LIN {X 0,Y 204.724,Z 772.28,A -85,B 0,C 180,E1 -21058.033,E2 -21058.033} C_VEL
LIN {X 0,Y 204.875,Z 767.063,A -85,B 0,C 180,E1 -21060.983,E2 -21060.983} C_VEL
LIN {X 0,Y 205.148,Z 761.459,A -85,B 0,C 180,E1 -21063.437,E2 -21063.437} C_VEL
LIN {X 0,Y 205.482,Z 754.231,A -85,B 0,C 180,E1 -21065.889,E2 -21065.889} C_VEL
LIN {X 0,Y 205.8,Z 746.691,A -85,B 0,C 180,E1 -21067.962,E2 -21067.962} C_VEL
LIN {X 0,Y 206.336,Z 737.426,A -85,B 0,C 180,E1 -21070.053,E2 -21070.053} C_VEL
LIN {X 0,Y 206.914,Z 727.818,A -85,B 0,C 180,E1 -21071.759,E2 -21071.759} C_VEL
LIN {X 0,Y 207.533,Z 717.475,A -85,B 0,C 180,E1 -21073.214,E2 -21073.214} C_VEL
LIN {X 0,Y 208.014,Z 706.264,A -85,B 0,C 180,E1 -21074.429,E2 -21074.429} C_VEL
LIN {X 0,Y 208.451,Z 692.158,A -85,B 0,C 180,E1 -21075.46,E2 -21075.46} C_VEL
LIN {X 0,Y 209.728,Z 644.97,A -85,B 0,C 180,E1 -21078.295,E2 -21078.295} C_VEL
LIN {X 0,Y 208.127,Z 622.961,A -85,B 0,C 180,E1 -21079.605,E2 -21079.605} C_VEL
LIN {X 0,Y 208.064,Z 617.38,A -85,B 0,C 180,E1 -21079.999,E2 -21079.999} C_VEL
LIN {X 0,Y 210.025,Z 597.2,A -85,B 0,C 180,E1 -21085.376,E2 -21085.376} C_VEL
LIN {X 0,Y 211.523,Z 584.285,A -85,B 0,C 180,E1 -21088.801,E2 -21088.801} C_VEL
LIN {X 0,Y 211.615,Z 582.311,A -85,B 0,C 180,E1 -21089.332,E2 -21089.332} C_VEL
LIN {X 0,Y 207.961,Z 564.134,A -85,B 0,C 180,E1 -21094.49,E2 -21094.49} C_VEL
LIN {X 0,Y 206.873,Z 558.873,A -85,B 0,C 180,E1 -21096.097,E2 -21096.097} C_VEL
LIN {X 0,Y 206.676,Z 558.686,A -85,B 0,C 180,E1 -21100.248,E2 -21100.248} C_VEL
LIN {X 0,Y 206.636,Z 558.719,A -85,B 0,C 180,E1 -21105.581,E2 -21105.581} C_VEL
LIN {X 0,Y 206.669,Z 558.926,A -85,B 0,C 180,E1 -21108.36,E2 -21108.36} C_VEL
LIN {X 0,Y 206.993,Z 560.154,A -85,B 0,C 180,E1 -21108.764,E2 -21108.764} C_VEL
LIN {X 0,Y 208.656,Z 562.795,A -85,B 0,C 180,E1 -21109.302,E2 -21109.302} C_VEL
LIN {X 0,Y 209.688,Z 564.185,A -85,B 0,C 180,E1 -21109.608,E2 -21109.608} C_VEL
LIN {X 0,Y 217.052,Z 575.841,A -85,B 0,C 180,E1 -21111.739,E2 -21111.739} C_VEL
LIN {X 0,Y 223.541,Z 588.628,A -85,B 0,C 180,E1 -21113.553,E2 -21113.553} C_VEL
LIN {X 0,Y 229.847,Z 603.206,A -85,B 0,C 180,E1 -21115.261,E2 -21115.261} C_VEL
LIN {X 0,Y 230.908,Z 606.056,A -85,B 0,C 180,E1 -21115.551,E2 -21115.551} C_VEL
LIN {X 0,Y 228.358,Z 664.194,A -85,B 0,C 180,E1 -21117.332,E2 -21117.332} C_VEL
LIN {X 0,Y 227.04,Z 677.769,A -85,B 0,C 180,E1 -21118.087,E2 -21118.087} C_VEL
LIN {X 0,Y 225.244,Z 690.404,A -85,B 0,C 180,E1 -21119.143,E2 -21119.143} C_VEL
LIN {X 0,Y 223.064,Z 702.192,A -85,B 0,C 180,E1 -21120.507,E2 -21120.507} C_VEL
LIN {X 0,Y 220.496,Z 713.529,A -85,B 0,C 180,E1 -21122.214,E2 -21122.214} C_VEL
LIN {X 0,Y 217.847,Z 723.743,A -85,B 0,C 180,E1 -21124.18,E2 -21124.18} C_VEL
LIN {X 0,Y 215.4,Z 732.864,A -85,B 0,C 180,E1 -21126.428,E2 -21126.428} C_VEL
LIN {X 0,Y 212.502,Z 741.807,A -85,B 0,C 180,E1 -21129.173,E2 -21129.173} C_VEL
LIN {X 0,Y 210.099,Z 748.972,A -85,B 0,C 180,E1 -21131.974,E2 -21131.974} C_VEL
LIN {X 0,Y 208.48,Z 753.802,A -85,B 0,C 180,E1 -21134.353,E2 -21134.353} C_VEL
LIN {X 0,Y 206.851,Z 758.495,A -85,B 0,C 180,E1 -21137.24,E2 -21137.24} C_VEL
LIN {X 0,Y 205.728,Z 762.077,A -85,B 0,C 180,E1 -21140.164,E2 -21140.164} C_VEL
LIN {X 0,Y 205.202,Z 763.927,A -85,B 0,C 180,E1 -21142.124,E2 -21142.124} C_VEL
LIN {X 0,Y 204.775,Z 765.519,A -85,B 0,C 180,E1 -21144.445,E2 -21144.445} C_VEL
LIN {X 0,Y 204.5,Z 766.916,A -85,B 0,C 180,E1 -21148.029,E2 -21148.029} C_VEL
LIN {X 0,Y 204.499,Z 767.144,A -85,B 0,C 180,E1 -21149.998,E2 -21149.998} C_VEL
LIN {X 0,Y 204.499,Z 766.951,A -85,B 0,C 180,E1 -21151.968,E2 -21151.968} C_VEL
LIN {X 0,Y 204.773,Z 765.603,A -85,B 0,C 180,E1 -21155.551,E2 -21155.551} C_VEL
LIN {X 0,Y 205.2,Z 764.046,A -85,B 0,C 180,E1 -21157.872,E2 -21157.872} C_VEL
LIN {X 0,Y 206.039,Z 761.177,A -85,B 0,C 180,E1 -21160.811,E2 -21160.811} C_VEL
LIN {X 0,Y 207.303,Z 757.284,A -85,B 0,C 180,E1 -21163.726,E2 -21163.726} C_VEL
LIN {X 0,Y 209.022,Z 752.264,A -85,B 0,C 180,E1 -21166.605,E2 -21166.605} C_VEL
LIN {X 0,Y 211.15,Z 745.94,A -85,B 0,C 180,E1 -21169.44,E2 -21169.44} C_VEL
LIN {X 0,Y 213.861,Z 738.019,A -85,B 0,C 180,E1 -21172.203,E2 -21172.203} C_VEL
LIN {X 0,Y 216.152,Z 730.125,A -85,B 0,C 180,E1 -21174.439,E2 -21174.439} C_VEL
LIN {X 0,Y 218.883,Z 720.101,A -85,B 0,C 180,E1 -21176.711,E2 -21176.711} C_VEL
LIN {X 0,Y 221.635,Z 709.007,A -85,B 0,C 180,E1 -21178.658,E2 -21178.658} C_VEL
LIN {X 0,Y 224.044,Z 698.121,A -85,B 0,C 180,E1 -21180.124,E2 -21180.124} C_VEL
LIN {X 0,Y 226.034,Z 686.085,A -85,B 0,C 180,E1 -21181.384,E2 -21181.384} C_VEL
LIN {X 0,Y 227.663,Z 673.169,A -85,B 0,C 180,E1 -21182.342,E2 -21182.342} C_VEL
LIN {X 0,Y 228.776,Z 659.415,A -85,B 0,C 180,E1 -21182.971,E2 -21182.971} C_VEL
LIN {X 0,Y 231.03,Z 606.183,A -85,B 0,C 180,E1 -21184.57,E2 -21184.57} C_VEL
LIN {X 0,Y 225.138,Z 592.104,A -85,B 0,C 180,E1 -21186.161,E2 -21186.161} C_VEL
LIN {X 0,Y 217.878,Z 577.227,A -85,B 0,C 180,E1 -21188.189,E2 -21188.189} C_VEL
LIN {X 0,Y 211.372,Z 566.808,A -85,B 0,C 180,E1 -21190.051,E2 -21190.051} C_VEL
LIN {X 0,Y 208.94,Z 563.085,A -85,B 0,C 180,E1 -21190.784,E2 -21190.784} C_VEL
LIN {X 0,Y 207.22,Z 560.726,A -85,B 0,C 180,E1 -21191.305,E2 -21191.305} C_VEL
LIN {X 0,Y 206.643,Z 558.739,A -85,B 0,C 180,E1 -21191.562,E2 -21191.562} C_VEL
LIN {X 0,Y 206.656,Z 558.72,A -85,B 0,C 180,E1 -21195.573,E2 -21195.573} C_VEL
LIN {X 0,Y 206.699,Z 558.712,A -85,B 0,C 180,E1 -21199.757,E2 -21199.757} C_VEL
LIN {X 0,Y 206.719,Z 558.701,A -85,B 0,C 180,E1 -21202.268,E2 -21202.268} C_VEL
LIN {X 0,Y 206.705,Z 558.728,A -85,B 0,C 180,E1 -21207.043,E2 -21207.043} C_VEL
LIN {X 0,Y 206.761,Z 558.716,A -85,B 0,C 180,E1 -21212.095,E2 -21212.095} C_VEL
LIN {X 0,Y 206.78,Z 558.717,A -85,B 0,C 180,E1 -21216.583,E2 -21216.583} C_VEL
LIN {X 0,Y 206.87,Z 558.707,A -85,B 0,C 180,E1 -21222.196,E2 -21222.196} C_VEL
LIN {X 0,Y 206.907,Z 558.71,A -85,B 0,C 180,E1 -21226.245,E2 -21226.245} C_VEL
LIN {X 0,Y 207.099,Z 558.667,A -85,B 0,C 180,E1 -21230.231,E2 -21230.231} C_VEL
LIN {X 0,Y 207.172,Z 558.672,A -85,B 0,C 180,E1 -21232.201,E2 -21232.201} C_VEL
LIN {X 0,Y 207.377,Z 558.637,A -85,B 0,C 180,E1 -21238.058,E2 -21238.058} C_VEL
LIN {X 0,Y 207.513,Z 558.637,A -85,B 0,C 180,E1 -21240,E2 -21240} C_VEL
LIN {X 0,Y 207.081,Z 558.67,A -85,B 0,C 180,E1 -21243.892,E2 -21243.892} C_VEL
LIN {X 0,Y 207.182,Z 558.674,A -85,B 0,C 180,E1 -21247.798,E2 -21247.798} C_VEL
LIN {X 0,Y 206.977,Z 558.693,A -85,B 0,C 180,E1 -21251.755,E2 -21251.755} C_VEL
LIN {X 0,Y 206.86,Z 558.701,A -85,B 0,C 180,E1 -21255.771,E2 -21255.771} C_VEL
LIN {X 0,Y 206.794,Z 558.723,A -85,B 0,C 180,E1 -21259.868,E2 -21259.868} C_VEL
LIN {X 0,Y 206.758,Z 558.732,A -85,B 0,C 180,E1 -21264.073,E2 -21264.073} C_VEL
LIN {X 0,Y 206.731,Z 558.734,A -85,B 0,C 180,E1 -21268.421,E2 -21268.421} C_VEL
LIN {X 0,Y 206.695,Z 558.729,A -85,B 0,C 180,E1 -21271.075,E2 -21271.075} C_VEL
LIN {X 0,Y 206.05,Z 558.819,A -85,B 0,C 180,E1 -21272.703,E2 -21272.703} C_VEL
LIN {X 0,Y 203.254,Z 559.173,A -85,B 0,C 180,E1 -21275.362,E2 -21275.362} C_VEL
LIN {X 0,Y 199.998,Z 559.573,A -85,B 0,C 180,E1 -21278.655,E2 -21278.655} C_VEL
LIN {X 0,Y 199.629,Z 559.607,A -85,B 0,C 180,E1 -21279.797,E2 -21279.797} C_VEL
LIN {X 0,Y 199.665,Z 559.81,A -85,B 0,C 180,E1 -21283.274,E2 -21283.274} C_VEL
LIN {X 0,Y 201.361,Z 565.661,A -85,B 0,C 180,E1 -21286.98,E2 -21286.98} C_VEL
LIN {X 0,Y 203.872,Z 570.229,A -85,B 0,C 180,E1 -21287.939,E2 -21287.939} C_VEL
LIN {X 0,Y 209.554,Z 580.484,A -85,B 0,C 180,E1 -21289.769,E2 -21289.769} C_VEL
LIN {X 0,Y 215.497,Z 592.713,A -85,B 0,C 180,E1 -21291.594,E2 -21291.594} C_VEL
LIN {X 0,Y 221.774,Z 607.31,A -85,B 0,C 180,E1 -21293.438,E2 -21293.438} C_VEL
LIN {X 0,Y 222.893,Z 610.664,A -85,B 0,C 180,E1 -21293.781,E2 -21293.781} C_VEL
LIN {X 0,Y 224.53,Z 623.993,A -85,B 0,C 180,E1 -21294.597,E2 -21294.597} C_VEL
LIN {X 0,Y 222.139,Z 674.383,A -85,B 0,C 180,E1 -21296.153,E2 -21296.153} C_VEL
LIN {X 0,Y 220.753,Z 687.704,A -85,B 0,C 180,E1 -21296.876,E2 -21296.876} C_VEL
LIN {X 0,Y 218.746,Z 699.995,A -85,B 0,C 180,E1 -21297.853,E2 -21297.853} C_VEL
LIN {X 0,Y 216.331,Z 712.2,A -85,B 0,C 180,E1 -21299.227,E2 -21299.227} C_VEL
LIN {X 0,Y 213.511,Z 723.759,A -85,B 0,C 180,E1 -21300.956,E2 -21300.956} C_VEL
LIN {X 0,Y 210.62,Z 734.171,A -85,B 0,C 180,E1 -21302.96,E2 -21302.96} C_VEL
LIN {X 0,Y 208.015,Z 742.689,A -85,B 0,C 180,E1 -21305.021,E2 -21305.021} C_VEL
LIN {X 0,Y 205.094,Z 751.926,A -85,B 0,C 180,E1 -21307.858,E2 -21307.858} C_VEL
LIN {X 0,Y 202.534,Z 759.353,A -85,B 0,C 180,E1 -21310.754,E2 -21310.754} C_VEL
LIN {X 0,Y 200.516,Z 765.318,A -85,B 0,C 180,E1 -21313.718,E2 -21313.718} C_VEL
LIN {X 0,Y 199.003,Z 770.036,A -85,B 0,C 180,E1 -21316.731,E2 -21316.731} C_VEL
LIN {X 0,Y 198.024,Z 773.649,A -85,B 0,C 180,E1 -21319.78,E2 -21319.78} C_VEL
LIN {X 0,Y 197.589,Z 775.512,A -85,B 0,C 180,E1 -21321.822,E2 -21321.822} C_VEL
LIN {X 0,Y 197.34,Z 776.909,A -85,B 0,C 180,E1 -21323.869,E2 -21323.869} C_VEL
LIN {X 0,Y 197.235,Z 778.517,A -85,B 0,C 180,E1 -21327.96,E2 -21327.96} C_VEL
LIN {X 0,Y 197.324,Z 778.731,A -85,B 0,C 180,E1 -21330.002,E2 -21330.002} C_VEL
LIN {X 0,Y 197.586,Z 777.91,A -85,B 0,C 180,E1 -21334.081,E2 -21334.081} C_VEL
LIN {X 0,Y 197.728,Z 777.713,A -85,B 0,C 180,E1 -21335.054,E2 -21335.054} C_VEL
LIN {X 0,Y 198.017,Z 780.538,A -85,B 0,C 180,E1 -21338.163,E2 -21338.163} C_VEL
LIN {X 0,Y 198.49,Z 781.851,A -85,B 0,C 180,E1 -21340.199,E2 -21340.199} C_VEL
LIN {X 0,Y 199.342,Z 782.728,A -85,B 0,C 180,E1 -21342.214,E2 -21342.214} C_VEL
LIN {X 0,Y 200.485,Z 783.034,A -85,B 0,C 180,E1 -21344.206,E2 -21344.206} C_VEL
LIN {X 0,Y 201.844,Z 782.917,A -85,B 0,C 180,E1 -21346.175,E2 -21346.175} C_VEL
LIN {X 0,Y 203.512,Z 782.403,A -85,B 0,C 180,E1 -21348.109,E2 -21348.109} C_VEL
LIN {X 0,Y 205.451,Z 781.417,A -85,B 0,C 180,E1 -21350.005,E2 -21350.005} C_VEL
LIN {X 0,Y 207.791,Z 779.883,A -85,B 0,C 180,E1 -21351.843,E2 -21351.843} C_VEL
LIN {X 0,Y 211.761,Z 776.762,A -85,B 0,C 180,E1 -21354.512,E2 -21354.512} C_VEL
LIN {X 0,Y 216.271,Z 772.492,A -85,B 0,C 180,E1 -21357.063,E2 -21357.063} C_VEL
LIN {X 0,Y 221.228,Z 766.817,A -85,B 0,C 180,E1 -21359.5,E2 -21359.5} C_VEL
LIN {X 0,Y 225.774,Z 761.035,A -85,B 0,C 180,E1 -21361.428,E2 -21361.428} C_VEL
LIN {X 0,Y 230.741,Z 753.954,A -85,B 0,C 180,E1 -21363.249,E2 -21363.249} C_VEL
LIN {X 0,Y 237.102,Z 743.44,A -85,B 0,C 180,E1 -21365.312,E2 -21365.312} C_VEL
LIN {X 0,Y 241.579,Z 734.691,A -85,B 0,C 180,E1 -21366.613,E2 -21366.613} C_VEL
LIN {X 0,Y 246.923,Z 722.426,A -85,B 0,C 180,E1 -21367.99,E2 -21367.99} C_VEL
LIN {X 0,Y 250.544,Z 711.991,A -85,B 0,C 180,E1 -21368.878,E2 -21368.878} C_VEL
LIN {X 0,Y 253.907,Z 699.571,A -85,B 0,C 180,E1 -21369.671,E2 -21369.671} C_VEL
LIN {X 0,Y 264.218,Z 655.621,A -85,B 0,C 180,E1 -21371.86,E2 -21371.86} C_VEL
LIN {X 0,Y 263.304,Z 655.908,A -85,B 0,C 180,E1 -21374.547,E2 -21374.547} C_VEL
LIN {X 0,Y 263.125,Z 657.91,A -85,B 0,C 180,E1 -21376.983,E2 -21376.983} C_VEL
LIN {X 0,Y 263.073,Z 660.384,A -85,B 0,C 180,E1 -21378.363,E2 -21378.363} C_VEL
LIN {X 0,Y 261.534,Z 671.304,A -85,B 0,C 180,E1 -21380.165,E2 -21380.165} C_VEL
LIN {X 0,Y 261.156,Z 673.713,A -85,B 0,C 180,E1 -21380.484,E2 -21380.484} C_VEL
LIN {X 0,Y 254.218,Z 704.594,A -85,B 0,C 180,E1 -21382.032,E2 -21382.032} C_VEL
LIN {X 0,Y 251.003,Z 715.292,A -85,B 0,C 180,E1 -21382.736,E2 -21382.736} C_VEL
LIN {X 0,Y 246.63,Z 726.648,A -85,B 0,C 180,E1 -21383.751,E2 -21383.751} C_VEL
LIN {X 0,Y 242.573,Z 735.584,A -85,B 0,C 180,E1 -21384.808,E2 -21384.808} C_VEL
LIN {X 0,Y 236.977,Z 745.877,A -85,B 0,C 180,E1 -21386.394,E2 -21386.394} C_VEL
LIN {X 0,Y 232.483,Z 753.037,A -85,B 0,C 180,E1 -21387.829,E2 -21387.829} C_VEL
LIN {X 0,Y 227.923,Z 759.399,A -85,B 0,C 180,E1 -21389.418,E2 -21389.418} C_VEL
LIN {X 0,Y 222.249,Z 766.367,A -85,B 0,C 180,E1 -21391.684,E2 -21391.684} C_VEL
LIN {X 0,Y 217.093,Z 771.721,A -85,B 0,C 180,E1 -21394.085,E2 -21394.085} C_VEL
LIN {X 0,Y 212.498,Z 775.684,A -85,B 0,C 180,E1 -21396.617,E2 -21396.617} C_VEL
LIN {X 0,Y 209.772,Z 777.732,A -85,B 0,C 180,E1 -21398.375,E2 -21398.375} C_VEL
LIN {X 0,Y 207.306,Z 779.257,A -85,B 0,C 180,E1 -21400.183,E2 -21400.183} C_VEL
LIN {X 0,Y 204.988,Z 780.219,A -85,B 0,C 180,E1 -21402.027,E2 -21402.027} C_VEL
LIN {X 0,Y 203.095,Z 780.735,A -85,B 0,C 180,E1 -21403.929,E2 -21403.929} C_VEL
LIN {X 0,Y 201.488,Z 780.83,A -85,B 0,C 180,E1 -21405.868,E2 -21405.868} C_VEL
LIN {X 0,Y 200.176,Z 780.459,A -85,B 0,C 180,E1 -21407.839,E2 -21407.839} C_VEL
LIN {X 0,Y 199.187,Z 779.534,A -85,B 0,C 180,E1 -21409.839,E2 -21409.839} C_VEL
LIN {X 0,Y 197.998,Z 776.571,A -85,B 0,C 180,E1 -21413.664,E2 -21413.664} C_VEL
LIN {X 0,Y 197.776,Z 772.563,A -85,B 0,C 180,E1 -21416.945,E2 -21416.945} C_VEL
LIN {X 0,Y 197.839,Z 767.433,A -85,B 0,C 180,E1 -21420,E2 -21420} C_VEL
LIN {X 0,Y 198.188,Z 760.658,A -85,B 0,C 180,E1 -21423.049,E2 -21423.049} C_VEL
LIN {X 0,Y 198.52,Z 753.348,A -85,B 0,C 180,E1 -21425.587,E2 -21425.587} C_VEL
LIN {X 0,Y 198.807,Z 746.178,A -85,B 0,C 180,E1 -21427.621,E2 -21427.621} C_VEL
LIN {X 0,Y 199.343,Z 736.407,A -85,B 0,C 180,E1 -21429.871,E2 -21429.871} C_VEL
LIN {X 0,Y 199.944,Z 726.35,A -85,B 0,C 180,E1 -21431.661,E2 -21431.661} C_VEL
LIN {X 0,Y 200.545,Z 715.701,A -85,B 0,C 180,E1 -21433.167,E2 -21433.167} C_VEL
LIN {X 0,Y 200.998,Z 704.275,A -85,B 0,C 180,E1 -21434.362,E2 -21434.362} C_VEL
LIN {X 0,Y 201.469,Z 690.665,A -85,B 0,C 180,E1 -21435.361,E2 -21435.361} C_VEL
LIN {X 0,Y 202.583,Z 644.705,A -85,B 0,C 180,E1 -21438.28,E2 -21438.28} C_VEL
LIN {X 0,Y 201.055,Z 621.901,A -85,B 0,C 180,E1 -21439.694,E2 -21439.694} C_VEL
LIN {X 0,Y 200.983,Z 617.432,A -85,B 0,C 180,E1 -21440.031,E2 -21440.031} C_VEL
LIN {X 0,Y 202.887,Z 598.036,A -85,B 0,C 180,E1 -21445.342,E2 -21445.342} C_VEL
LIN {X 0,Y 204.541,Z 583.598,A -85,B 0,C 180,E1 -21449.28,E2 -21449.28} C_VEL
LIN {X 0,Y 201.511,Z 568.102,A -85,B 0,C 180,E1 -21453.768,E2 -21453.768} C_VEL
LIN {X 0,Y 199.833,Z 559.742,A -85,B 0,C 180,E1 -21456.34,E2 -21456.34} C_VEL
LIN {X 0,Y 199.649,Z 559.577,A -85,B 0,C 180,E1 -21459.319,E2 -21459.319} C_VEL
LIN {X 0,Y 199.582,Z 559.577,A -85,B 0,C 180,E1 -21464.771,E2 -21464.771} C_VEL
LIN {X 0,Y 199.628,Z 559.896,A -85,B 0,C 180,E1 -21466.634,E2 -21466.634} C_VEL
LIN {X 0,Y 199.926,Z 561.099,A -85,B 0,C 180,E1 -21466.997,E2 -21466.997} C_VEL
LIN {X 0,Y 201.612,Z 563.736,A -85,B 0,C 180,E1 -21467.588,E2 -21467.588} C_VEL
LIN {X 0,Y 202.681,Z 565.024,A -85,B 0,C 180,E1 -21467.926,E2 -21467.926} C_VEL
LIN {X 0,Y 205.037,Z 568.479,A -85,B 0,C 180,E1 -21468.681,E2 -21468.681} C_VEL
LIN {X 0,Y 212.911,Z 581.152,A -85,B 0,C 180,E1 -21471.074,E2 -21471.074} C_VEL
LIN {X 0,Y 219.766,Z 595.203,A -85,B 0,C 180,E1 -21473.081,E2 -21473.081} C_VEL
LIN {X 0,Y 225.024,Z 607.901,A -85,B 0,C 180,E1 -21474.579,E2 -21474.579} C_VEL
LIN {X 0,Y 222.433,Z 664.277,A -85,B 0,C 180,E1 -21476.34,E2 -21476.34} C_VEL
LIN {X 0,Y 221.049,Z 678.056,A -85,B 0,C 180,E1 -21477.121,E2 -21477.121} C_VEL
LIN {X 0,Y 219.191,Z 690.615,A -85,B 0,C 180,E1 -21478.193,E2 -21478.193} C_VEL
LIN {X 0,Y 216.911,Z 702.402,A -85,B 0,C 180,E1 -21479.584,E2 -21479.584} C_VEL
LIN {X 0,Y 214.258,Z 713.738,A -85,B 0,C 180,E1 -21481.331,E2 -21481.331} C_VEL
LIN {X 0,Y 211.475,Z 723.952,A -85,B 0,C 180,E1 -21483.341,E2 -21483.341} C_VEL
LIN {X 0,Y 208.809,Z 733.344,A -85,B 0,C 180,E1 -21485.726,E2 -21485.726} C_VEL
LIN {X 0,Y 205.887,Z 742.014,A -85,B 0,C 180,E1 -21488.47,E2 -21488.47} C_VEL
LIN {X 0,Y 203.363,Z 749.178,A -85,B 0,C 180,E1 -21491.355,E2 -21491.355} C_VEL
LIN {X 0,Y 201.639,Z 754.008,A -85,B 0,C 180,E1 -21493.808,E2 -21493.808} C_VEL
LIN {X 0,Y 199.942,Z 758.7,A -85,B 0,C 180,E1 -21496.791,E2 -21496.791} C_VEL
LIN {X 0,Y 198.741,Z 762.283,A -85,B 0,C 180,E1 -21499.814,E2 -21499.814} C_VEL
LIN {X 0,Y 198.164,Z 764.133,A -85,B 0,C 180,E1 -21501.843,E2 -21501.843} C_VEL
LIN {X 0,Y 197.671,Z 765.903,A -85,B 0,C 180,E1 -21504.575,E2 -21504.575} C_VEL
LIN {X 0,Y 197.407,Z 767.121,A -85,B 0,C 180,E1 -21507.958,E2 -21507.958} C_VEL
LIN {X 0,Y 197.401,Z 767.348,A -85,B 0,C 180,E1 -21509.998,E2 -21509.998} C_VEL
LIN {X 0,Y 197.406,Z 767.155,A -85,B 0,C 180,E1 -21512.038,E2 -21512.038} C_VEL
LIN {X 0,Y 197.669,Z 765.987,A -85,B 0,C 180,E1 -21515.419,E2 -21515.419} C_VEL
LIN {X 0,Y 198.162,Z 764.25,A -85,B 0,C 180,E1 -21518.154,E2 -21518.154} C_VEL
LIN {X 0,Y 199.056,Z 761.381,A -85,B 0,C 180,E1 -21521.195,E2 -21521.195} C_VEL
LIN {X 0,Y 200.419,Z 757.487,A -85,B 0,C 180,E1 -21524.207,E2 -21524.207} C_VEL
LIN {X 0,Y 202.212,Z 752.468,A -85,B 0,C 180,E1 -21527.181,E2 -21527.181} C_VEL
LIN {X 0,Y 204.465,Z 746.143,A -85,B 0,C 180,E1 -21530.102,E2 -21530.102} C_VEL
LIN {X 0,Y 207.302,Z 738.221,A -85,B 0,C 180,E1 -21532.945,E2 -21532.945} C_VEL
LIN {X 0,Y 209.92,Z 729.627,A -85,B 0,C 180,E1 -21535.424,E2 -21535.424} C_VEL
LIN {X 0,Y 212.575,Z 720.302,A -85,B 0,C 180,E1 -21537.57,E2 -21537.57} C_VEL
LIN {X 0,Y 215.456,Z 709.206,A -85,B 0,C 180,E1 -21539.56,E2 -21539.56} C_VEL
LIN {X 0,Y 217.939,Z 698.32,A -85,B 0,C 180,E1 -21541.06,E2 -21541.06} C_VEL
LIN {X 0,Y 220.023,Z 686.281,A -85,B 0,C 180,E1 -21542.344,E2 -21542.344} C_VEL
LIN {X 0,Y 221.662,Z 673.728,A -85,B 0,C 180,E1 -21543.302,E2 -21543.302} C_VEL
LIN {X 0,Y 222.799,Z 660.906,A -85,B 0,C 180,E1 -21543.915,E2 -21543.915} C_VEL
LIN {X 0,Y 225.154,Z 608.112,A -85,B 0,C 180,E1 -21545.54,E2 -21545.54} C_VEL
LIN {X 0,Y 219.131,Z 593.764,A -85,B 0,C 180,E1 -21547.258,E2 -21547.258} C_VEL
LIN {X 0,Y 212.451,Z 580.214,A -85,B 0,C 180,E1 -21549.229,E2 -21549.229} C_VEL
LIN {X 0,Y 204.883,Z 568.339,A -85,B 0,C 180,E1 -21551.534,E2 -21551.534} C_VEL
LIN {X 0,Y 202.682,Z 565.022,A -85,B 0,C 180,E1 -21552.247,E2 -21552.247} C_VEL
LIN {X 0,Y 200.158,Z 561.683,A -85,B 0,C 180,E1 -21553.072,E2 -21553.072} C_VEL
LIN {X 0,Y 199.577,Z 559.608,A -85,B 0,C 180,E1 -21553.388,E2 -21553.388} C_VEL
LIN {X 0,Y 199.616,Z 559.621,A -85,B 0,C 180,E1 -21558.014,E2 -21558.014} C_VEL
LIN {X 0,Y 199.673,Z 559.577,A -85,B 0,C 180,E1 -21560.742,E2 -21560.742} C_VEL
LIN {X 0,Y 199.631,Z 559.619,A -85,B 0,C 180,E1 -21565.717,E2 -21565.717} C_VEL
LIN {X 0,Y 199.699,Z 559.6,A -85,B 0,C 180,E1 -21568.136,E2 -21568.136} C_VEL
LIN {X 0,Y 199.681,Z 559.598,A -85,B 0,C 180,E1 -21572.771,E2 -21572.771} C_VEL
LIN {X 0,Y 199.732,Z 559.59,A -85,B 0,C 180,E1 -21577.228,E2 -21577.228} C_VEL
LIN {X 0,Y 199.832,Z 559.587,A -85,B 0,C 180,E1 -21581.721,E2 -21581.721} C_VEL
LIN {X 0,Y 199.842,Z 559.584,A -85,B 0,C 180,E1 -21585.749,E2 -21585.749} C_VEL
LIN {X 0,Y 200.064,Z 559.543,A -85,B 0,C 180,E1 -21589.884,E2 -21589.884} C_VEL
LIN {X 0,Y 200.033,Z 559.567,A -85,B 0,C 180,E1 -21593.95,E2 -21593.95} C_VEL
LIN {X 0,Y 200.316,Z 559.515,A -85,B 0,C 180,E1 -21597.989,E2 -21597.989} C_VEL
LIN {X 0,Y 200.477,Z 559.514,A -85,B 0,C 180,E1 -21600,E2 -21600} C_VEL
LIN {X 0,Y 200.026,Z 559.549,A -85,B 0,C 180,E1 -21604.029,E2 -21604.029} C_VEL
LIN {X 0,Y 200.126,Z 559.552,A -85,B 0,C 180,E1 -21608.075,E2 -21608.075} C_VEL
LIN {X 0,Y 199.909,Z 559.577,A -85,B 0,C 180,E1 -21612.177,E2 -21612.177} C_VEL
LIN {X 0,Y 199.799,Z 559.58,A -85,B 0,C 180,E1 -21616.344,E2 -21616.344} C_VEL
LIN {X 0,Y 199.818,Z 559.594,A -85,B 0,C 180,E1 -21618.454,E2 -21618.454} C_VEL
LIN {X 0,Y 199.731,Z 559.605,A -85,B 0,C 180,E1 -21623.818,E2 -21623.818} C_VEL
LIN {X 0,Y 199.702,Z 559.608,A -85,B 0,C 180,E1 -21628.385,E2 -21628.385} C_VEL
LIN {X 0,Y 199.666,Z 559.611,A -85,B 0,C 180,E1 -21632.356,E2 -21632.356} C_VEL
LIN {X 0,Y 199.639,Z 559.584,A -85,B 0,C 180,E1 -21636.76,E2 -21636.76} C_VEL
LIN {X 0,Y 199.629,Z 559.607,A -85,B 0,C 180,E1 -21639.797,E2 -21639.797} C_VEL
LIN {X 0,Y 199.366,Z 560.017,A -85,B 0,C 180,E1 -21640.883,E2 -21640.883} C_VEL
LIN {X 0,Y 198.566,Z 561.868,A -85,B 0,C 180,E1 -21642.437,E2 -21642.437} C_VEL
LIN {X 0,Y 197.596,Z 565.883,A -85,B 0,C 180,E1 -21644.333,E2 -21644.333} C_VEL
LIN {X 0,Y 197.588,Z 569.644,A -85,B 0,C 180,E1 -21645.619,E2 -21645.619} C_VEL
LIN {X 0,Y 198.808,Z 573.68,A -85,B 0,C 180,E1 -21646.739,E2 -21646.739} C_VEL
LIN {X 0,Y 199.595,Z 575.018,A -85,B 0,C 180,E1 -21647.059,E2 -21647.059} C_VEL
LIN {X 0,Y 205,Z 584.884,A -85,B 0,C 180,E1 -21648.89,E2 -21648.89} C_VEL
LIN {X 0,Y 210.673,Z 596.819,A -85,B 0,C 180,E1 -21650.73,E2 -21650.73} C_VEL
LIN {X 0,Y 216.727,Z 611.181,A -85,B 0,C 180,E1 -21652.607,E2 -21652.607} C_VEL
LIN {X 0,Y 217.406,Z 613.832,A -85,B 0,C 180,E1 -21652.85,E2 -21652.85} C_VEL
LIN {X 0,Y 218.712,Z 625.371,A -85,B 0,C 180,E1 -21653.568,E2 -21653.568} C_VEL
LIN {X 0,Y 216.205,Z 675.122,A -85,B 0,C 180,E1 -21655.149,E2 -21655.149} C_VEL
LIN {X 0,Y 214.635,Z 688.965,A -85,B 0,C 180,E1 -21655.939,E2 -21655.939} C_VEL
LIN {X 0,Y 212.57,Z 700.904,A -85,B 0,C 180,E1 -21656.942,E2 -21656.942} C_VEL
LIN {X 0,Y 210.25,Z 712,A -85,B 0,C 180,E1 -21658.235,E2 -21658.235} C_VEL
LIN {X 0,Y 207.331,Z 723.558,A -85,B 0,C 180,E1 -21660.003,E2 -21660.003} C_VEL
LIN {X 0,Y 204.305,Z 733.969,A -85,B 0,C 180,E1 -21662.053,E2 -21662.053} C_VEL
LIN {X 0,Y 201.562,Z 742.486,A -85,B 0,C 180,E1 -21664.163,E2 -21664.163} C_VEL
LIN {X 0,Y 198.507,Z 751.722,A -85,B 0,C 180,E1 -21667.082,E2 -21667.082} C_VEL
LIN {X 0,Y 195.81,Z 759.148,A -85,B 0,C 180,E1 -21670.066,E2 -21670.066} C_VEL
LIN {X 0,Y 193.67,Z 765.114,A -85,B 0,C 180,E1 -21673.126,E2 -21673.126} C_VEL
LIN {X 0,Y 192.051,Z 769.831,A -85,B 0,C 180,E1 -21676.241,E2 -21676.241} C_VEL
LIN {X 0,Y 191.013,Z 773.445,A -85,B 0,C 180,E1 -21679.401,E2 -21679.401} C_VEL
LIN {X 0,Y 190.538,Z 775.307,A -85,B 0,C 180,E1 -21681.517,E2 -21681.517} C_VEL
LIN {X 0,Y 190.278,Z 776.705,A -85,B 0,C 180,E1 -21683.64,E2 -21683.64} C_VEL
LIN {X 0,Y 190.144,Z 778.312,A -85,B 0,C 180,E1 -21687.884,E2 -21687.884} C_VEL
LIN {X 0,Y 190.229,Z 778.526,A -85,B 0,C 180,E1 -21690.002,E2 -21690.002} C_VEL
LIN {X 0,Y 190.299,Z 778.303,A -85,B 0,C 180,E1 -21692.118,E2 -21692.118} C_VEL
LIN {X 0,Y 190.78,Z 777.167,A -85,B 0,C 180,E1 -21695.809,E2 -21695.809} C_VEL
LIN {X 0,Y 191.041,Z 779.709,A -85,B 0,C 180,E1 -21698.464,E2 -21698.464} C_VEL
LIN {X 0,Y 191.528,Z 781.216,A -85,B 0,C 180,E1 -21700.574,E2 -21700.574} C_VEL
LIN {X 0,Y 193.596,Z 782.806,A -85,B 0,C 180,E1 -21704.723,E2 -21704.723} C_VEL
LIN {X 0,Y 195.039,Z 783.008,A -85,B 0,C 180,E1 -21706.756,E2 -21706.756} C_VEL
LIN {X 0,Y 196.774,Z 782.668,A -85,B 0,C 180,E1 -21708.752,E2 -21708.752} C_VEL
LIN {X 0,Y 198.809,Z 781.887,A -85,B 0,C 180,E1 -21710.704,E2 -21710.704} C_VEL
LIN {X 0,Y 201.262,Z 780.695,A -85,B 0,C 180,E1 -21712.591,E2 -21712.591} C_VEL
LIN {X 0,Y 205.422,Z 777.989,A -85,B 0,C 180,E1 -21715.321,E2 -21715.321} C_VEL
LIN {X 0,Y 210.133,Z 774.156,A -85,B 0,C 180,E1 -21717.922,E2 -21717.922} C_VEL
LIN {X 0,Y 215.34,Z 769.183,A -85,B 0,C 180,E1 -21720.391,E2 -21720.391} C_VEL
LIN {X 0,Y 221.069,Z 762.779,A -85,B 0,C 180,E1 -21722.716,E2 -21722.716} C_VEL
LIN {X 0,Y 227.385,Z 754.633,A -85,B 0,C 180,E1 -21724.877,E2 -21724.877} C_VEL
LIN {X 0,Y 232.995,Z 746.259,A -85,B 0,C 180,E1 -21726.567,E2 -21726.567} C_VEL
LIN {X 0,Y 238.877,Z 735.963,A -85,B 0,C 180,E1 -21728.16,E2 -21728.16} C_VEL
LIN {X 0,Y 243.222,Z 726.986,A -85,B 0,C 180,E1 -21729.206,E2 -21729.206} C_VEL
LIN {X 0,Y 248.316,Z 714.263,A -85,B 0,C 180,E1 -21730.349,E2 -21730.349} C_VEL
LIN {X 0,Y 251.67,Z 703.464,A -85,B 0,C 180,E1 -21731.063,E2 -21731.063} C_VEL
LIN {X 0,Y 261.822,Z 662.666,A -85,B 0,C 180,E1 -21733.101,E2 -21733.101} C_VEL
LIN {X 0,Y 261.442,Z 662.914,A -85,B 0,C 180,E1 -21734.773,E2 -21734.773} C_VEL
LIN {X 0,Y 261.227,Z 664.498,A -85,B 0,C 180,E1 -21736.587,E2 -21736.587} C_VEL
LIN {X 0,Y 261.158,Z 665.955,A -85,B 0,C 180,E1 -21737.416,E2 -21737.416} C_VEL
LIN {X 0,Y 259.44,Z 675.625,A -85,B 0,C 180,E1 -21739.004,E2 -21739.004} C_VEL
LIN {X 0,Y 252.531,Z 704.506,A -85,B 0,C 180,E1 -21740.46,E2 -21740.46} C_VEL
LIN {X 0,Y 249.154,Z 715.25,A -85,B 0,C 180,E1 -21741.126,E2 -21741.126} C_VEL
LIN {X 0,Y 244.573,Z 726.615,A -85,B 0,C 180,E1 -21742.104,E2 -21742.104} C_VEL
LIN {X 0,Y 240.215,Z 735.617,A -85,B 0,C 180,E1 -21743.146,E2 -21743.146} C_VEL
LIN {X 0,Y 234.196,Z 746.074,A -85,B 0,C 180,E1 -21744.713,E2 -21744.713} C_VEL
LIN {X 0,Y 228.54,Z 754.378,A -85,B 0,C 180,E1 -21746.39,E2 -21746.39} C_VEL
LIN {X 0,Y 222.153,Z 762.427,A -85,B 0,C 180,E1 -21748.534,E2 -21748.534} C_VEL
LIN {X 0,Y 216.257,Z 768.627,A -85,B 0,C 180,E1 -21750.825,E2 -21750.825} C_VEL
LIN {X 0,Y 210.877,Z 773.426,A -85,B 0,C 180,E1 -21753.261,E2 -21753.261} C_VEL
LIN {X 0,Y 206.102,Z 777.003,A -85,B 0,C 180,E1 -21755.846,E2 -21755.846} C_VEL
LIN {X 0,Y 203.244,Z 778.655,A -85,B 0,C 180,E1 -21757.643,E2 -21757.643} C_VEL
LIN {X 0,Y 200.67,Z 779.883,A -85,B 0,C 180,E1 -21759.499,E2 -21759.499} C_VEL
LIN {X 0,Y 198.281,Z 780.69,A -85,B 0,C 180,E1 -21761.397,E2 -21761.397} C_VEL
LIN {X 0,Y 196.295,Z 780.963,A -85,B 0,C 180,E1 -21763.356,E2 -21763.356} C_VEL
LIN {X 0,Y 194.615,Z 780.731,A -85,B 0,C 180,E1 -21765.358,E2 -21765.358} C_VEL
LIN {X 0,Y 193.264,Z 780.092,A -85,B 0,C 180,E1 -21767.397,E2 -21767.397} C_VEL
LIN {X 0,Y 192.224,Z 779.042,A -85,B 0,C 180,E1 -21769.467,E2 -21769.467} C_VEL
LIN {X 0,Y 191.52,Z 777.463,A -85,B 0,C 180,E1 -21771.56,E2 -21771.56} C_VEL
LIN {X 0,Y 190.84,Z 773.857,A -85,B 0,C 180,E1 -21774.952,E2 -21774.952} C_VEL
LIN {X 0,Y 190.798,Z 769.554,A -85,B 0,C 180,E1 -21777.889,E2 -21777.889} C_VEL
LIN {X 0,Y 191.043,Z 763.529,A -85,B 0,C 180,E1 -21781.054,E2 -21781.054} C_VEL
LIN {X 0,Y 191.337,Z 757.07,A -85,B 0,C 180,E1 -21783.686,E2 -21783.686} C_VEL
LIN {X 0,Y 191.687,Z 748.878,A -85,B 0,C 180,E1 -21786.315,E2 -21786.315} C_VEL
LIN {X 0,Y 192.114,Z 740.762,A -85,B 0,C 180,E1 -21788.414,E2 -21788.414} C_VEL
LIN {X 0,Y 192.649,Z 730.818,A -85,B 0,C 180,E1 -21790.51,E2 -21790.51} C_VEL
LIN {X 0,Y 193.312,Z 719.597,A -85,B 0,C 180,E1 -21792.333,E2 -21792.333} C_VEL
LIN {X 0,Y 193.777,Z 709.118,A -85,B 0,C 180,E1 -21793.636,E2 -21793.636} C_VEL
LIN {X 0,Y 194.167,Z 695.751,A -85,B 0,C 180,E1 -21794.811,E2 -21794.811} C_VEL
LIN {X 0,Y 195.568,Z 645.972,A -85,B 0,C 180,E1 -21798.124,E2 -21798.124} C_VEL
LIN {X 0,Y 193.973,Z 622.735,A -85,B 0,C 180,E1 -21799.639,E2 -21799.639} C_VEL
LIN {X 0,Y 193.909,Z 617.344,A -85,B 0,C 180,E1 -21800.068,E2 -21800.068} C_VEL
LIN {X 0,Y 195.995,Z 596.44,A -85,B 0,C 180,E1 -21805.968,E2 -21805.968} C_VEL
LIN {X 0,Y 197.426,Z 583.506,A -85,B 0,C 180,E1 -21809.599,E2 -21809.599} C_VEL
LIN {X 0,Y 193.848,Z 565.909,A -85,B 0,C 180,E1 -21814.849,E2 -21814.849} C_VEL
LIN {X 0,Y 192.767,Z 560.648,A -85,B 0,C 180,E1 -21816.537,E2 -21816.537} C_VEL
LIN {X 0,Y 192.528,Z 560.435,A -85,B 0,C 180,E1 -21821.077,E2 -21821.077} C_VEL
LIN {X 0,Y 192.566,Z 560.729,A -85,B 0,C 180,E1 -21824.586,E2 -21824.586} C_VEL
LIN {X 0,Y 192.91,Z 561.952,A -85,B 0,C 180,E1 -21825.048,E2 -21825.048} C_VEL
LIN {X 0,Y 194.518,Z 564.593,A -85,B 0,C 180,E1 -21825.676,E2 -21825.676} C_VEL
LIN {X 0,Y 195.709,Z 565.917,A -85,B 0,C 180,E1 -21826.085,E2 -21826.085} C_VEL
LIN {X 0,Y 197.971,Z 569.344,A -85,B 0,C 180,E1 -21826.884,E2 -21826.884} C_VEL
LIN {X 0,Y 203.881,Z 578.29,A -85,B 0,C 180,E1 -21828.845,E2 -21828.845} C_VEL
LIN {X 0,Y 209.039,Z 586.997,A -85,B 0,C 180,E1 -21830.461,E2 -21830.461} C_VEL
LIN {X 0,Y 215.42,Z 600.593,A -85,B 0,C 180,E1 -21832.424,E2 -21832.424} C_VEL
LIN {X 0,Y 219.227,Z 609.816,A -85,B 0,C 180,E1 -21833.561,E2 -21833.561} C_VEL
LIN {X 0,Y 216.573,Z 664.5,A -85,B 0,C 180,E1 -21835.302,E2 -21835.302} C_VEL
LIN {X 0,Y 215.13,Z 678.348,A -85,B 0,C 180,E1 -21836.103,E2 -21836.103} C_VEL
LIN {X 0,Y 213.196,Z 690.827,A -85,B 0,C 180,E1 -21837.188,E2 -21837.188} C_VEL
LIN {X 0,Y 210.819,Z 702.612,A -85,B 0,C 180,E1 -21838.607,E2 -21838.607} C_VEL
LIN {X 0,Y 208.071,Z 713.946,A -85,B 0,C 180,E1 -21840.395,E2 -21840.395} C_VEL
LIN {X 0,Y 205.167,Z 724.159,A -85,B 0,C 180,E1 -21842.454,E2 -21842.454} C_VEL
LIN {X 0,Y 202.255,Z 733.806,A -85,B 0,C 180,E1 -21844.972,E2 -21844.972} C_VEL
LIN {X 0,Y 199.31,Z 742.22,A -85,B 0,C 180,E1 -21847.723,E2 -21847.723} C_VEL
LIN {X 0,Y 196.655,Z 749.385,A -85,B 0,C 180,E1 -21850.695,E2 -21850.695} C_VEL
LIN {X 0,Y 194.823,Z 754.215,A -85,B 0,C 180,E1 -21853.225,E2 -21853.225} C_VEL
LIN {X 0,Y 193.033,Z 758.906,A -85,B 0,C 180,E1 -21856.309,E2 -21856.309} C_VEL
LIN {X 0,Y 191.748,Z 762.489,A -85,B 0,C 180,E1 -21859.438,E2 -21859.438} C_VEL
LIN {X 0,Y 191.127,Z 764.339,A -85,B 0,C 180,E1 -21861.54,E2 -21861.54} C_VEL
LIN {X 0,Y 190.569,Z 766.285,A -85,B 0,C 180,E1 -21864.709,E2 -21864.709} C_VEL
LIN {X 0,Y 190.317,Z 767.326,A -85,B 0,C 180,E1 -21867.882,E2 -21867.882} C_VEL
LIN {X 0,Y 190.306,Z 767.553,A -85,B 0,C 180,E1 -21869.998,E2 -21869.998} C_VEL
LIN {X 0,Y 190.316,Z 767.36,A -85,B 0,C 180,E1 -21872.114,E2 -21872.114} C_VEL
LIN {X 0,Y 190.721,Z 765.81,A -85,B 0,C 180,E1 -21876.345,E2 -21876.345} C_VEL
LIN {X 0,Y 191.125,Z 764.455,A -85,B 0,C 180,E1 -21878.456,E2 -21878.456} C_VEL
LIN {X 0,Y 192.098,Z 761.585,A -85,B 0,C 180,E1 -21881.606,E2 -21881.606} C_VEL
LIN {X 0,Y 193.538,Z 757.691,A -85,B 0,C 180,E1 -21884.724,E2 -21884.724} C_VEL
LIN {X 0,Y 195.431,Z 752.671,A -85,B 0,C 180,E1 -21887.797,E2 -21887.797} C_VEL
LIN {X 0,Y 197.816,Z 746.345,A -85,B 0,C 180,E1 -21890.809,E2 -21890.809} C_VEL
LIN {X 0,Y 200.779,Z 738.423,A -85,B 0,C 180,E1 -21893.735,E2 -21893.735} C_VEL
LIN {X 0,Y 203.427,Z 730.126,A -85,B 0,C 180,E1 -21896.204,E2 -21896.204} C_VEL
LIN {X 0,Y 206.322,Z 720.502,A -85,B 0,C 180,E1 -21898.48,E2 -21898.48} C_VEL
LIN {X 0,Y 209.328,Z 709.406,A -85,B 0,C 180,E1 -21900.516,E2 -21900.516} C_VEL
LIN {X 0,Y 211.888,Z 698.519,A -85,B 0,C 180,E1 -21902.05,E2 -21902.05} C_VEL
LIN {X 0,Y 214.074,Z 686.478,A -85,B 0,C 180,E1 -21903.358,E2 -21903.358} C_VEL
LIN {X 0,Y 215.815,Z 673.548,A -85,B 0,C 180,E1 -21904.357,E2 -21904.357} C_VEL
LIN {X 0,Y 217.016,Z 659.969,A -85,B 0,C 180,E1 -21905.001,E2 -21905.001} C_VEL
LIN {X 0,Y 219.345,Z 610.04,A -85,B 0,C 180,E1 -21906.561,E2 -21906.561} C_VEL
LIN {X 0,Y 213.093,Z 595.306,A -85,B 0,C 180,E1 -21908.446,E2 -21908.446} C_VEL
LIN {X 0,Y 207.573,Z 584.161,A -85,B 0,C 180,E1 -21910.168,E2 -21910.168} C_VEL
LIN {X 0,Y 200.593,Z 573.18,A -85,B 0,C 180,E1 -21912.405,E2 -21912.405} C_VEL
LIN {X 0,Y 197.382,Z 568.631,A -85,B 0,C 180,E1 -21913.491,E2 -21913.491} C_VEL
LIN {X 0,Y 195.174,Z 565.175,A -85,B 0,C 180,E1 -21914.288,E2 -21914.288} C_VEL
LIN {X 0,Y 193.221,Z 562.727,A -85,B 0,C 180,E1 -21914.985,E2 -21914.985} C_VEL
LIN {X 0,Y 192.56,Z 560.474,A -85,B 0,C 180,E1 -21915.352,E2 -21915.352} C_VEL
LIN {X 0,Y 192.571,Z 560.467,A -85,B 0,C 180,E1 -21920.029,E2 -21920.029} C_VEL
LIN {X 0,Y 192.597,Z 560.486,A -85,B 0,C 180,E1 -21924.278,E2 -21924.278} C_VEL
LIN {X 0,Y 192.603,Z 560.492,A -85,B 0,C 180,E1 -21929.279,E2 -21929.279} C_VEL
LIN {X 0,Y 192.659,Z 560.474,A -85,B 0,C 180,E1 -21931.691,E2 -21931.691} C_VEL
LIN {X 0,Y 192.7,Z 560.472,A -85,B 0,C 180,E1 -21936.348,E2 -21936.348} C_VEL
LIN {X 0,Y 192.775,Z 560.468,A -85,B 0,C 180,E1 -21941.413,E2 -21941.413} C_VEL
LIN {X 0,Y 192.847,Z 560.462,A -85,B 0,C 180,E1 -21947.369,E2 -21947.369} C_VEL
LIN {X 0,Y 193.062,Z 560.422,A -85,B 0,C 180,E1 -21951.627,E2 -21951.627} C_VEL
LIN {X 0,Y 193.258,Z 560.394,A -85,B 0,C 180,E1 -21957.916,E2 -21957.916} C_VEL
LIN {X 0,Y 193.44,Z 560.39,A -85,B 0,C 180,E1 -21960,E2 -21960} C_VEL
LIN {X 0,Y 192.973,Z 560.427,A -85,B 0,C 180,E1 -21964.177,E2 -21964.177} C_VEL
LIN {X 0,Y 193.073,Z 560.426,A -85,B 0,C 180,E1 -21968.372,E2 -21968.372} C_VEL
LIN {X 0,Y 192.847,Z 560.462,A -85,B 0,C 180,E1 -21972.63,E2 -21972.63} C_VEL
LIN {X 0,Y 192.775,Z 560.472,A -85,B 0,C 180,E1 -21978.587,E2 -21978.587} C_VEL
LIN {X 0,Y 192.658,Z 560.488,A -85,B 0,C 180,E1 -21984.225,E2 -21984.225} C_VEL
LIN {X 0,Y 192.638,Z 560.491,A -85,B 0,C 180,E1 -21988.89,E2 -21988.89} C_VEL
LIN {X 0,Y 192.591,Z 560.497,A -85,B 0,C 180,E1 -21993.187,E2 -21993.187} C_VEL
LIN {X 0,Y 192.59,Z 560.474,A -85,B 0,C 180,E1 -21998.343,E2 -21998.343} C_VEL
LIN {X 0,Y 192.601,Z 560.624,A -85,B 0,C 180,E1 -22001.661,E2 -22001.661} C_VEL
LIN {X 0,Y 193.957,Z 565.253,A -85,B 0,C 180,E1 -22004.866,E2 -22004.866} C_VEL
LIN {X 0,Y 196.049,Z 569.224,A -85,B 0,C 180,E1 -22005.805,E2 -22005.805} C_VEL
LIN {X 0,Y 197.993,Z 572.347,A -85,B 0,C 180,E1 -22006.498,E2 -22006.498} C_VEL
LIN {X 0,Y 199.595,Z 575.018,A -85,B 0,C 180,E1 -22007.059,E2 -22007.059} C_VEL
LIN {X 0,Y 201.178,Z 578.024,A -85,B 0,C 180,E1 -22007.617,E2 -22007.617} C_VEL
LIN {X 0,Y 202.306,Z 581.444,A -85,B 0,C 180,E1 -22008.065,E2 -22008.065} C_VEL
LIN {X 0,Y 203.706,Z 588.897,A -85,B 0,C 180,E1 -22008.758,E2 -22008.758} C_VEL
LIN {X 0,Y 205.315,Z 598.44,A -85,B 0,C 180,E1 -22009.578,E2 -22009.578} C_VEL
LIN {X 0,Y 207.122,Z 603.667,A -85,B 0,C 180,E1 -22010.23,E2 -22010.23} C_VEL
LIN {X 0,Y 211.804,Z 615.318,A -85,B 0,C 180,E1 -22011.763,E2 -22011.763} C_VEL
LIN {X 0,Y 212.98,Z 626.15,A -85,B 0,C 180,E1 -22012.462,E2 -22012.462} C_VEL
LIN {X 0,Y 210.421,Z 674.981,A -85,B 0,C 180,E1 -22014.048,E2 -22014.048} C_VEL
LIN {X 0,Y 208.775,Z 688.887,A -85,B 0,C 180,E1 -22014.856,E2 -22014.856} C_VEL
LIN {X 0,Y 206.452,Z 701.712,A -85,B 0,C 180,E1 -22015.977,E2 -22015.977} C_VEL
LIN {X 0,Y 203.849,Z 713.384,A -85,B 0,C 180,E1 -22017.407,E2 -22017.407} C_VEL
LIN {X 0,Y 200.838,Z 724.651,A -85,B 0,C 180,E1 -22019.22,E2 -22019.22} C_VEL
LIN {X 0,Y 197.728,Z 734.802,A -85,B 0,C 180,E1 -22021.327,E2 -22021.327} C_VEL
LIN {X 0,Y 194.603,Z 743.953,A -85,B 0,C 180,E1 -22023.745,E2 -22023.745} C_VEL
LIN {X 0,Y 191.452,Z 752.962,A -85,B 0,C 180,E1 -22026.795,E2 -22026.795} C_VEL
LIN {X 0,Y 188.719,Z 760.06,A -85,B 0,C 180,E1 -22029.852,E2 -22029.852} C_VEL
LIN {X 0,Y 186.857,Z 764.909,A -85,B 0,C 180,E1 -22032.491,E2 -22032.491} C_VEL
LIN {X 0,Y 185.124,Z 769.626,A -85,B 0,C 180,E1 -22035.716,E2 -22035.716} C_VEL
LIN {X 0,Y 183.993,Z 773.239,A -85,B 0,C 180,E1 -22038.992,E2 -22038.992} C_VEL
LIN {X 0,Y 183.508,Z 775.102,A -85,B 0,C 180,E1 -22041.19,E2 -22041.19} C_VEL
LIN {X 0,Y 183.211,Z 776.5,A -85,B 0,C 180,E1 -22043.394,E2 -22043.394} C_VEL
LIN {X 0,Y 183.04,Z 778.107,A -85,B 0,C 180,E1 -22047.801,E2 -22047.801} C_VEL
LIN {X 0,Y 183.136,Z 778.321,A -85,B 0,C 180,E1 -22050.002,E2 -22050.002} C_VEL
LIN {X 0,Y 183.214,Z 778.098,A -85,B 0,C 180,E1 -22052.2,E2 -22052.2} C_VEL
LIN {X 0,Y 183.832,Z 776.616,A -85,B 0,C 180,E1 -22056.726,E2 -22056.726} C_VEL
LIN {X 0,Y 184.106,Z 778.629,A -85,B 0,C 180,E1 -22058.785,E2 -22058.785} C_VEL
LIN {X 0,Y 184.603,Z 780.332,A -85,B 0,C 180,E1 -22060.975,E2 -22060.975} C_VEL
LIN {X 0,Y 185.505,Z 781.647,A -85,B 0,C 180,E1 -22063.141,E2 -22063.141} C_VEL
LIN {X 0,Y 186.729,Z 782.512,A -85,B 0,C 180,E1 -22065.277,E2 -22065.277} C_VEL
LIN {X 0,Y 190.058,Z 782.783,A -85,B 0,C 180,E1 -22069.441,E2 -22069.441} C_VEL
LIN {X 0,Y 192.199,Z 782.353,A -85,B 0,C 180,E1 -22071.45,E2 -22071.45} C_VEL
LIN {X 0,Y 194.759,Z 781.397,A -85,B 0,C 180,E1 -22073.389,E2 -22073.389} C_VEL
LIN {X 0,Y 197.591,Z 779.971,A -85,B 0,C 180,E1 -22075.268,E2 -22075.268} C_VEL
LIN {X 0,Y 204.06,Z 775.852,A -85,B 0,C 180,E1 -22078.829,E2 -22078.829} C_VEL
LIN {X 0,Y 209.484,Z 771.327,A -85,B 0,C 180,E1 -22081.335,E2 -22081.335} C_VEL
LIN {X 0,Y 215.457,Z 765.571,A -85,B 0,C 180,E1 -22083.68,E2 -22083.68} C_VEL
LIN {X 0,Y 220.903,Z 759.57,A -85,B 0,C 180,E1 -22085.496,E2 -22085.496} C_VEL
LIN {X 0,Y 227.813,Z 750.821,A -85,B 0,C 180,E1 -22087.539,E2 -22087.539} C_VEL
LIN {X 0,Y 233.249,Z 742.612,A -85,B 0,C 180,E1 -22088.977,E2 -22088.977} C_VEL
LIN {X 0,Y 239.009,Z 732.739,A -85,B 0,C 180,E1 -22090.31,E2 -22090.31} C_VEL
LIN {X 0,Y 244.312,Z 721.591,A -85,B 0,C 180,E1 -22091.426,E2 -22091.426} C_VEL
LIN {X 0,Y 249.015,Z 709.33,A -85,B 0,C 180,E1 -22092.365,E2 -22092.365} C_VEL
LIN {X 0,Y 253.448,Z 693.667,A -85,B 0,C 180,E1 -22093.206,E2 -22093.206} C_VEL
LIN {X 0,Y 259.669,Z 669.593,A -85,B 0,C 180,E1 -22094.383,E2 -22094.383} C_VEL
LIN {X 0,Y 259.318,Z 671.328,A -85,B 0,C 180,E1 -22096.336,E2 -22096.336} C_VEL
LIN {X 0,Y 259.021,Z 672.884,A -85,B 0,C 180,E1 -22096.689,E2 -22096.689} C_VEL
LIN {X 0,Y 257.878,Z 678.405,A -85,B 0,C 180,E1 -22097.567,E2 -22097.567} C_VEL
LIN {X 0,Y 250.757,Z 706.286,A -85,B 0,C 180,E1 -22098.937,E2 -22098.937} C_VEL
LIN {X 0,Y 246.911,Z 717.41,A -85,B 0,C 180,E1 -22099.643,E2 -22099.643} C_VEL
LIN {X 0,Y 242.129,Z 728.243,A -85,B 0,C 180,E1 -22100.584,E2 -22100.584} C_VEL
LIN {X 0,Y 236.288,Z 739.197,A -85,B 0,C 180,E1 -22101.89,E2 -22101.89} C_VEL
LIN {X 0,Y 231.277,Z 747.076,A -85,B 0,C 180,E1 -22103.119,E2 -22103.119} C_VEL
LIN {X 0,Y 225.707,Z 754.632,A -85,B 0,C 180,E1 -22104.64,E2 -22104.64} C_VEL
LIN {X 0,Y 219.865,Z 761.623,A -85,B 0,C 180,E1 -22106.43,E2 -22106.43} C_VEL
LIN {X 0,Y 214.311,Z 767.27,A -85,B 0,C 180,E1 -22108.352,E2 -22108.352} C_VEL
LIN {X 0,Y 208.377,Z 772.361,A -85,B 0,C 180,E1 -22110.722,E2 -22110.722} C_VEL
LIN {X 0,Y 202.969,Z 776.186,A -85,B 0,C 180,E1 -22113.247,E2 -22113.247} C_VEL
LIN {X 0,Y 199.718,Z 778.102,A -85,B 0,C 180,E1 -22115.022,E2 -22115.022} C_VEL
LIN {X 0,Y 196.754,Z 779.575,A -85,B 0,C 180,E1 -22116.864,E2 -22116.864} C_VEL
LIN {X 0,Y 194.069,Z 780.479,A -85,B 0,C 180,E1 -22118.768,E2 -22118.768} C_VEL
LIN {X 0,Y 191.573,Z 780.927,A -85,B 0,C 180,E1 -22120.721,E2 -22120.721} C_VEL
LIN {X 0,Y 189.523,Z 780.975,A -85,B 0,C 180,E1 -22122.743,E2 -22122.743} C_VEL
LIN {X 0,Y 187.768,Z 780.591,A -85,B 0,C 180,E1 -22124.811,E2 -22124.811} C_VEL
LIN {X 0,Y 186.372,Z 779.665,A -85,B 0,C 180,E1 -22126.923,E2 -22126.923} C_VEL
LIN {X 0,Y 185.282,Z 778.301,A -85,B 0,C 180,E1 -22129.067,E2 -22129.067} C_VEL
LIN {X 0,Y 184.572,Z 776.521,A -85,B 0,C 180,E1 -22131.239,E2 -22131.239} C_VEL
LIN {X 0,Y 183.916,Z 772.67,A -85,B 0,C 180,E1 -22134.653,E2 -22134.653} C_VEL
LIN {X 0,Y 183.879,Z 767.912,A -85,B 0,C 180,E1 -22137.81,E2 -22137.81} C_VEL
LIN {X 0,Y 184.181,Z 761.498,A -85,B 0,C 180,E1 -22141.093,E2 -22141.093} C_VEL
LIN {X 0,Y 184.489,Z 754.541,A -85,B 0,C 180,E1 -22143.823,E2 -22143.823} C_VEL
LIN {X 0,Y 184.757,Z 747.721,A -85,B 0,C 180,E1 -22146.005,E2 -22146.005} C_VEL
LIN {X 0,Y 185.223,Z 738.734,A -85,B 0,C 180,E1 -22148.345,E2 -22148.345} C_VEL
LIN {X 0,Y 185.845,Z 727.567,A -85,B 0,C 180,E1 -22150.625,E2 -22150.625} C_VEL
LIN {X 0,Y 186.396,Z 717.356,A -85,B 0,C 180,E1 -22152.245,E2 -22152.245} C_VEL
LIN {X 0,Y 186.891,Z 706.386,A -85,B 0,C 180,E1 -22153.594,E2 -22153.594} C_VEL
LIN {X 0,Y 187.238,Z 692.698,A -85,B 0,C 180,E1 -22154.746,E2 -22154.746} C_VEL
LIN {X 0,Y 188.484,Z 646.28,A -85,B 0,C 180,E1 -22158.021,E2 -22158.021} C_VEL
LIN {X 0,Y 186.861,Z 623.211,A -85,B 0,C 180,E1 -22159.569,E2 -22159.569} C_VEL
LIN {X 0,Y 186.799,Z 617.47,A -85,B 0,C 180,E1 -22160.024,E2 -22160.024} C_VEL
LIN {X 0,Y 188.845,Z 597.178,A -85,B 0,C 180,E1 -22165.931,E2 -22165.931} C_VEL
LIN {X 0,Y 190.381,Z 584.515,A -85,B 0,C 180,E1 -22169.587,E2 -22169.587} C_VEL
LIN {X 0,Y 186.774,Z 566.606,A -85,B 0,C 180,E1 -22175.072,E2 -22175.072} C_VEL
LIN {X 0,Y 185.715,Z 561.532,A -85,B 0,C 180,E1 -22176.754,E2 -22176.754} C_VEL
LIN {X 0,Y 185.462,Z 561.428,A -85,B 0,C 180,E1 -22182.077,E2 -22182.077} C_VEL
LIN {X 0,Y 185.642,Z 562.325,A -85,B 0,C 180,E1 -22182.723,E2 -22182.723} C_VEL
LIN {X 0,Y 187.321,Z 565.311,A -85,B 0,C 180,E1 -22183.506,E2 -22183.506} C_VEL
LIN {X 0,Y 188.839,Z 566.896,A -85,B 0,C 180,E1 -22184.078,E2 -22184.078} C_VEL
LIN {X 0,Y 191.1,Z 570.295,A -85,B 0,C 180,E1 -22184.958,E2 -22184.958} C_VEL
LIN {X 0,Y 197.362,Z 579.494,A -85,B 0,C 180,E1 -22187.214,E2 -22187.214} C_VEL
LIN {X 0,Y 203.919,Z 590.294,A -85,B 0,C 180,E1 -22189.404,E2 -22189.404} C_VEL
LIN {X 0,Y 210.55,Z 604.654,A -85,B 0,C 180,E1 -22191.562,E2 -22191.562} C_VEL
LIN {X 0,Y 213.484,Z 611.779,A -85,B 0,C 180,E1 -22192.487,E2 -22192.487} C_VEL
LIN {X 0,Y 210.792,Z 664.786,A -85,B 0,C 180,E1 -22194.211,E2 -22194.211} C_VEL
LIN {X 0,Y 209.347,Z 678.093,A -85,B 0,C 180,E1 -22194.988,E2 -22194.988} C_VEL
LIN {X 0,Y 207.279,Z 691.037,A -85,B 0,C 180,E1 -22196.127,E2 -22196.127} C_VEL
LIN {X 0,Y 204.8,Z 702.822,A -85,B 0,C 180,E1 -22197.573,E2 -22197.573} C_VEL
LIN {X 0,Y 201.925,Z 714.155,A -85,B 0,C 180,E1 -22199.4,E2 -22199.4} C_VEL
LIN {X 0,Y 198.895,Z 724.368,A -85,B 0,C 180,E1 -22201.507,E2 -22201.507} C_VEL
LIN {X 0,Y 195.963,Z 733.431,A -85,B 0,C 180,E1 -22203.904,E2 -22203.904} C_VEL
LIN {X 0,Y 192.766,Z 742.427,A -85,B 0,C 180,E1 -22206.924,E2 -22206.924} C_VEL
LIN {X 0,Y 189.965,Z 749.591,A -85,B 0,C 180,E1 -22209.986,E2 -22209.986} C_VEL
LIN {X 0,Y 188.034,Z 754.421,A -85,B 0,C 180,E1 -22212.6,E2 -22212.6} C_VEL
LIN {X 0,Y 186.129,Z 759.112,A -85,B 0,C 180,E1 -22215.791,E2 -22215.791} C_VEL
LIN {X 0,Y 184.759,Z 762.695,A -85,B 0,C 180,E1 -22219.034,E2 -22219.034} C_VEL
LIN {X 0,Y 184.116,Z 764.544,A -85,B 0,C 180,E1 -22221.216,E2 -22221.216} C_VEL
LIN {X 0,Y 183.459,Z 766.665,A -85,B 0,C 180,E1 -22224.888,E2 -22224.888} C_VEL
LIN {X 0,Y 183.229,Z 767.53,A -85,B 0,C 180,E1 -22227.8,E2 -22227.8} C_VEL
LIN {X 0,Y 183.212,Z 767.757,A -85,B 0,C 180,E1 -22229.998,E2 -22229.998} C_VEL
LIN {X 0,Y 183.228,Z 767.564,A -85,B 0,C 180,E1 -22232.196,E2 -22232.196} C_VEL
LIN {X 0,Y 183.459,Z 766.722,A -85,B 0,C 180,E1 -22235.111,E2 -22235.111} C_VEL
LIN {X 0,Y 184.114,Z 764.659,A -85,B 0,C 180,E1 -22238.781,E2 -22238.781} C_VEL
LIN {X 0,Y 185.13,Z 761.789,A -85,B 0,C 180,E1 -22242.05,E2 -22242.05} C_VEL
LIN {X 0,Y 186.66,Z 757.895,A -85,B 0,C 180,E1 -22245.279,E2 -22245.279} C_VEL
LIN {X 0,Y 188.68,Z 752.875,A -85,B 0,C 180,E1 -22248.456,E2 -22248.456} C_VEL
LIN {X 0,Y 191.201,Z 746.548,A -85,B 0,C 180,E1 -22251.564,E2 -22251.564} C_VEL
LIN {X 0,Y 194.283,Z 738.626,A -85,B 0,C 180,E1 -22254.58,E2 -22254.58} C_VEL
LIN {X 0,Y 196.992,Z 730.589,A -85,B 0,C 180,E1 -22257.044,E2 -22257.044} C_VEL
LIN {X 0,Y 200.124,Z 720.703,A -85,B 0,C 180,E1 -22259.447,E2 -22259.447} C_VEL
LIN {X 0,Y 203.26,Z 709.605,A -85,B 0,C 180,E1 -22261.529,E2 -22261.529} C_VEL
LIN {X 0,Y 205.907,Z 698.718,A -85,B 0,C 180,E1 -22263.098,E2 -22263.098} C_VEL
LIN {X 0,Y 208.193,Z 686.675,A -85,B 0,C 180,E1 -22264.43,E2 -22264.43} C_VEL
LIN {X 0,Y 209.965,Z 674.138,A -85,B 0,C 180,E1 -22265.424,E2 -22265.424} C_VEL
LIN {X 0,Y 211.158,Z 661.562,A -85,B 0,C 180,E1 -22266.052,E2 -22266.052} C_VEL
LIN {X 0,Y 213.608,Z 611.989,A -85,B 0,C 180,E1 -22267.637,E2 -22267.637} C_VEL
LIN {X 0,Y 207.311,Z 597.265,A -85,B 0,C 180,E1 -22269.648,E2 -22269.648} C_VEL
LIN {X 0,Y 202.764,Z 588.171,A -85,B 0,C 180,E1 -22271.147,E2 -22271.147} C_VEL
LIN {X 0,Y 196.137,Z 577.725,A -85,B 0,C 180,E1 -22273.388,E2 -22273.388} C_VEL
LIN {X 0,Y 190.906,Z 570.059,A -85,B 0,C 180,E1 -22275.302,E2 -22275.302} C_VEL
LIN {X 0,Y 188.765,Z 566.688,A -85,B 0,C 180,E1 -22276.148,E2 -22276.148} C_VEL
LIN {X 0,Y 186.39,Z 564.056,A -85,B 0,C 180,E1 -22277.064,E2 -22277.064} C_VEL
LIN {X 0,Y 185.48,Z 561.378,A -85,B 0,C 180,E1 -22277.537,E2 -22277.537} C_VEL
LIN {X 0,Y 185.539,Z 561.34,A -85,B 0,C 180,E1 -22282.695,E2 -22282.695} C_VEL
LIN {X 0,Y 185.54,Z 561.363,A -85,B 0,C 180,E1 -22287.974,E2 -22287.974} C_VEL
LIN {X 0,Y 185.577,Z 561.366,A -85,B 0,C 180,E1 -22290.575,E2 -22290.575} C_VEL
LIN {X 0,Y 185.582,Z 561.367,A -85,B 0,C 180,E1 -22295.382,E2 -22295.382} C_VEL
LIN {X 0,Y 185.688,Z 561.353,A -85,B 0,C 180,E1 -22301.115,E2 -22301.115} C_VEL
LIN {X 0,Y 185.759,Z 561.345,A -85,B 0,C 180,E1 -22306.879,E2 -22306.879} C_VEL
LIN {X 0,Y 186.008,Z 561.297,A -85,B 0,C 180,E1 -22311.307,E2 -22311.307} C_VEL
LIN {X 0,Y 186.202,Z 561.271,A -85,B 0,C 180,E1 -22317.837,E2 -22317.837} C_VEL
LIN {X 0,Y 186.403,Z 561.267,A -85,B 0,C 180,E1 -22320,E2 -22320} C_VEL
LIN {X 0,Y 185.921,Z 561.306,A -85,B 0,C 180,E1 -22324.336,E2 -22324.336} C_VEL
LIN {X 0,Y 186.023,Z 561.3,A -85,B 0,C 180,E1 -22328.692,E2 -22328.692} C_VEL
LIN {X 0,Y 185.759,Z 561.346,A -85,B 0,C 180,E1 -22333.121,E2 -22333.121} C_VEL
LIN {X 0,Y 185.688,Z 561.355,A -85,B 0,C 180,E1 -22338.885,E2 -22338.885} C_VEL
LIN {X 0,Y 185.595,Z 561.367,A -85,B 0,C 180,E1 -22344.663,E2 -22344.663} C_VEL
LIN {X 0,Y 185.572,Z 561.368,A -85,B 0,C 180,E1 -22349.494,E2 -22349.494} C_VEL
LIN {X 0,Y 185.497,Z 561.358,A -85,B 0,C 180,E1 -22354.632,E2 -22354.632} C_VEL
LIN {X 0,Y 185.528,Z 561.369,A -85,B 0,C 180,E1 -22359.383,E2 -22359.383} C_VEL
LIN {X 0,Y 185.558,Z 561.613,A -85,B 0,C 180,E1 -22360.081,E2 -22360.081} C_VEL
LIN {X 0,Y 186.6,Z 565.145,A -85,B 0,C 180,E1 -22362.607,E2 -22362.607} C_VEL
LIN {X 0,Y 189.385,Z 569.763,A -85,B 0,C 180,E1 -22363.852,E2 -22363.852} C_VEL
LIN {X 0,Y 193.781,Z 577.126,A -85,B 0,C 180,E1 -22365.555,E2 -22365.555} C_VEL
LIN {X 0,Y 200.007,Z 588.316,A -85,B 0,C 180,E1 -22367.801,E2 -22367.801} C_VEL
LIN {X 0,Y 206.652,Z 602.541,A -85,B 0,C 180,E1 -22370.073,E2 -22370.073} C_VEL
LIN {X 0,Y 207.122,Z 603.667,A -85,B 0,C 180,E1 -22370.23,E2 -22370.23} C_VEL
LIN {X 0,Y 208.308,Z 607.073,A -85,B 0,C 180,E1 -22370.648,E2 -22370.648} C_VEL
LIN {X 0,Y 209.005,Z 612.758,A -85,B 0,C 180,E1 -22371.049,E2 -22371.049} C_VEL
LIN {X 0,Y 208.784,Z 618.687,A -85,B 0,C 180,E1 -22371.257,E2 -22371.257} C_VEL
LIN {X 0,Y 206.912,Z 635.218,A -85,B 0,C 180,E1 -22371.561,E2 -22371.561} C_VEL
LIN {X 0,Y 204.714,Z 674.929,A -85,B 0,C 180,E1 -22372.891,E2 -22372.891} C_VEL
LIN {X 0,Y 203.005,Z 688.81,A -85,B 0,C 180,E1 -22373.714,E2 -22373.714} C_VEL
LIN {X 0,Y 200.624,Z 701.514,A -85,B 0,C 180,E1 -22374.845,E2 -22374.845} C_VEL
LIN {X 0,Y 197.913,Z 713.184,A -85,B 0,C 180,E1 -22376.302,E2 -22376.302} C_VEL
LIN {X 0,Y 194.775,Z 724.45,A -85,B 0,C 180,E1 -22378.152,E2 -22378.152} C_VEL
LIN {X 0,Y 191.502,Z 734.6,A -85,B 0,C 180,E1 -22380.304,E2 -22380.304} C_VEL
LIN {X 0,Y 188.237,Z 743.75,A -85,B 0,C 180,E1 -22382.785,E2 -22382.785} C_VEL
LIN {X 0,Y 185.243,Z 751.873,A -85,B 0,C 180,E1 -22385.581,E2 -22385.581} C_VEL
LIN {X 0,Y 182.496,Z 758.742,A -85,B 0,C 180,E1 -22388.542,E2 -22388.542} C_VEL
LIN {X 0,Y 180.077,Z 764.705,A -85,B 0,C 180,E1 -22391.809,E2 -22391.809} C_VEL
LIN {X 0,Y 178.199,Z 769.421,A -85,B 0,C 180,E1 -22395.148,E2 -22395.148} C_VEL
LIN {X 0,Y 176.999,Z 773.035,A -85,B 0,C 180,E1 -22398.551,E2 -22398.551} C_VEL
LIN {X 0,Y 176.467,Z 774.898,A -85,B 0,C 180,E1 -22400.836,E2 -22400.836} C_VEL
LIN {X 0,Y 176.139,Z 776.295,A -85,B 0,C 180,E1 -22403.127,E2 -22403.127} C_VEL
LIN {X 0,Y 175.949,Z 777.903,A -85,B 0,C 180,E1 -22407.713,E2 -22407.713} C_VEL
LIN {X 0,Y 176.044,Z 778.117,A -85,B 0,C 180,E1 -22410.002,E2 -22410.002} C_VEL
LIN {X 0,Y 176.132,Z 777.893,A -85,B 0,C 180,E1 -22412.289,E2 -22412.289} C_VEL
LIN {X 0,Y 176.577,Z 776.851,A -85,B 0,C 180,E1 -22415.711,E2 -22415.711} C_VEL
LIN {X 0,Y 176.993,Z 776.017,A -85,B 0,C 180,E1 -22417.703,E2 -22417.703} C_VEL
LIN {X 0,Y 177.689,Z 779.434,A -85,B 0,C 180,E1 -22421.408,E2 -22421.408} C_VEL
LIN {X 0,Y 178.65,Z 780.907,A -85,B 0,C 180,E1 -22423.655,E2 -22423.655} C_VEL
LIN {X 0,Y 181.488,Z 782.596,A -85,B 0,C 180,E1 -22428.049,E2 -22428.049} C_VEL
LIN {X 0,Y 183.372,Z 782.84,A -85,B 0,C 180,E1 -22430.18,E2 -22430.18} C_VEL
LIN {X 0,Y 185.614,Z 782.558,A -85,B 0,C 180,E1 -22432.251,E2 -22432.251} C_VEL
LIN {X 0,Y 191.244,Z 780.862,A -85,B 0,C 180,E1 -22436.169,E2 -22436.169} C_VEL
LIN {X 0,Y 196.197,Z 778.353,A -85,B 0,C 180,E1 -22438.922,E2 -22438.922} C_VEL
LIN {X 0,Y 201.72,Z 774.764,A -85,B 0,C 180,E1 -22441.509,E2 -22441.509} C_VEL
LIN {X 0,Y 207.737,Z 770.055,A -85,B 0,C 180,E1 -22443.934,E2 -22443.934} C_VEL
LIN {X 0,Y 214.316,Z 764.063,A -85,B 0,C 180,E1 -22446.178,E2 -22446.178} C_VEL
LIN {X 0,Y 221.426,Z 756.412,A -85,B 0,C 180,E1 -22448.239,E2 -22448.239} C_VEL
LIN {X 0,Y 227.661,Z 748.578,A -85,B 0,C 180,E1 -22449.835,E2 -22449.835} C_VEL
LIN {X 0,Y 233.241,Z 740.493,A -85,B 0,C 180,E1 -22451.123,E2 -22451.123} C_VEL
LIN {X 0,Y 239.662,Z 729.535,A -85,B 0,C 180,E1 -22452.414,E2 -22452.414} C_VEL
LIN {X 0,Y 244.527,Z 719.403,A -85,B 0,C 180,E1 -22453.331,E2 -22453.331} C_VEL
LIN {X 0,Y 249.176,Z 707.28,A -85,B 0,C 180,E1 -22454.145,E2 -22454.145} C_VEL
LIN {X 0,Y 254.92,Z 687.257,A -85,B 0,C 180,E1 -22455.166,E2 -22455.166} C_VEL
LIN {X 0,Y 257.438,Z 677.989,A -85,B 0,C 180,E1 -22455.573,E2 -22455.573} C_VEL
LIN {X 0,Y 256.622,Z 681.195,A -85,B 0,C 180,E1 -22456.092,E2 -22456.092} C_VEL
LIN {X 0,Y 250.059,Z 705.846,A -85,B 0,C 180,E1 -22457.278,E2 -22457.278} C_VEL
LIN {X 0,Y 246.189,Z 716.725,A -85,B 0,C 180,E1 -22457.923,E2 -22457.923} C_VEL
LIN {X 0,Y 241.279,Z 727.376,A -85,B 0,C 180,E1 -22458.775,E2 -22458.775} C_VEL
LIN {X 0,Y 235.833,Z 737.467,A -85,B 0,C 180,E1 -22459.876,E2 -22459.876} C_VEL
LIN {X 0,Y 229.875,Z 746.483,A -85,B 0,C 180,E1 -22461.189,E2 -22461.189} C_VEL
LIN {X 0,Y 223.538,Z 754.673,A -85,B 0,C 180,E1 -22462.755,E2 -22462.755} C_VEL
LIN {X 0,Y 217.483,Z 761.43,A -85,B 0,C 180,E1 -22464.432,E2 -22464.432} C_VEL
LIN {X 0,Y 211.147,Z 767.457,A -85,B 0,C 180,E1 -22466.429,E2 -22466.429} C_VEL
LIN {X 0,Y 204.348,Z 772.813,A -85,B 0,C 180,E1 -22468.943,E2 -22468.943} C_VEL
LIN {X 0,Y 198.56,Z 776.525,A -85,B 0,C 180,E1 -22471.456,E2 -22471.456} C_VEL
LIN {X 0,Y 193.376,Z 779.121,A -85,B 0,C 180,E1 -22474.143,E2 -22474.143} C_VEL
LIN {X 0,Y 190.279,Z 780.204,A -85,B 0,C 180,E1 -22476.028,E2 -22476.028} C_VEL
LIN {X 0,Y 187.506,Z 780.902,A -85,B 0,C 180,E1 -22477.987,E2 -22477.987} C_VEL
LIN {X 0,Y 184.901,Z 781.156,A -85,B 0,C 180,E1 -22479.996,E2 -22479.996} C_VEL
LIN {X 0,Y 180.947,Z 780.168,A -85,B 0,C 180,E1 -22484.224,E2 -22484.224} C_VEL
LIN {X 0,Y 179.5,Z 779.088,A -85,B 0,C 180,E1 -22486.413,E2 -22486.413} C_VEL
LIN {X 0,Y 177.957,Z 776.533,A -85,B 0,C 180,E1 -22489.763,E2 -22489.763} C_VEL
LIN {X 0,Y 177.1,Z 772.857,A -85,B 0,C 180,E1 -22493.163,E2 -22493.163} C_VEL
LIN {X 0,Y 177,Z 768.028,A -85,B 0,C 180,E1 -22496.586,E2 -22496.586} C_VEL
LIN {X 0,Y 177.2,Z 761.753,A -85,B 0,C 180,E1 -22500,E2 -22500} C_VEL
LIN {X 0,Y 177.55,Z 754.916,A -85,B 0,C 180,E1 -22502.836,E2 -22502.836} C_VEL
LIN {X 0,Y 177.839,Z 748.229,A -85,B 0,C 180,E1 -22505.101,E2 -22505.101} C_VEL
LIN {X 0,Y 178.155,Z 740.278,A -85,B 0,C 180,E1 -22507.326,E2 -22507.326} C_VEL
LIN {X 0,Y 178.657,Z 730.951,A -85,B 0,C 180,E1 -22509.476,E2 -22509.476} C_VEL
LIN {X 0,Y 179.262,Z 719.916,A -85,B 0,C 180,E1 -22511.433,E2 -22511.433} C_VEL
LIN {X 0,Y 179.747,Z 709.523,A -85,B 0,C 180,E1 -22512.848,E2 -22512.848} C_VEL
LIN {X 0,Y 180.09,Z 696.664,A -85,B 0,C 180,E1 -22514.117,E2 -22514.117} C_VEL
LIN {X 0,Y 181.407,Z 646.625,A -85,B 0,C 180,E1 -22517.837,E2 -22517.837} C_VEL
LIN {X 0,Y 179.801,Z 622.674,A -85,B 0,C 180,E1 -22519.537,E2 -22519.537} C_VEL
LIN {X 0,Y 179.721,Z 617.369,A -85,B 0,C 180,E1 -22520.011,E2 -22520.011} C_VEL
LIN {X 0,Y 182.143,Z 594.237,A -85,B 0,C 180,E1 -22526.961,E2 -22526.961} C_VEL
LIN {X 0,Y 183.247,Z 585.492,A -85,B 0,C 180,E1 -22529.559,E2 -22529.559} C_VEL
LIN {X 0,Y 180.289,Z 570.316,A -85,B 0,C 180,E1 -22534.315,E2 -22534.315} C_VEL
LIN {X 0,Y 178.663,Z 562.488,A -85,B 0,C 180,E1 -22536.912,E2 -22536.912} C_VEL
LIN {X 0,Y 178.46,Z 562.283,A -85,B 0,C 180,E1 -22539.422,E2 -22539.422} C_VEL
LIN {X 0,Y 178.575,Z 562.889,A -85,B 0,C 180,E1 -22540.125,E2 -22540.125} C_VEL
LIN {X 0,Y 180.002,Z 565.846,A -85,B 0,C 180,E1 -22541.004,E2 -22541.004} C_VEL
LIN {X 0,Y 181.889,Z 567.746,A -85,B 0,C 180,E1 -22541.799,E2 -22541.799} C_VEL
LIN {X 0,Y 184.217,Z 571.286,A -85,B 0,C 180,E1 -22542.809,E2 -22542.809} C_VEL
LIN {X 0,Y 185.565,Z 573.08,A -85,B 0,C 180,E1 -22543.36,E2 -22543.36} C_VEL
LIN {X 0,Y 192.965,Z 583.931,A -85,B 0,C 180,E1 -22546.209,E2 -22546.209} C_VEL
LIN {X 0,Y 199.432,Z 594.737,A -85,B 0,C 180,E1 -22548.491,E2 -22548.491} C_VEL
LIN {X 0,Y 205.676,Z 608.633,A -85,B 0,C 180,E1 -22550.644,E2 -22550.644} C_VEL
LIN {X 0,Y 207.781,Z 613.817,A -85,B 0,C 180,E1 -22551.348,E2 -22551.348} C_VEL
LIN {X 0,Y 205.163,Z 664.335,A -85,B 0,C 180,E1 -22553.024,E2 -22553.024} C_VEL
LIN {X 0,Y 203.709,Z 677.362,A -85,B 0,C 180,E1 -22553.774,E2 -22553.774} C_VEL
LIN {X 0,Y 201.647,Z 690.167,A -85,B 0,C 180,E1 -22554.893,E2 -22554.893} C_VEL
LIN {X 0,Y 199.282,Z 701.449,A -85,B 0,C 180,E1 -22556.257,E2 -22556.257} C_VEL
LIN {X 0,Y 196.203,Z 713.077,A -85,B 0,C 180,E1 -22558.104,E2 -22558.104} C_VEL
LIN {X 0,Y 193.019,Z 723.52,A -85,B 0,C 180,E1 -22560.256,E2 -22560.256} C_VEL
LIN {X 0,Y 190.086,Z 732.256,A -85,B 0,C 180,E1 -22562.542,E2 -22562.542} C_VEL
LIN {X 0,Y 187.372,Z 739.901,A -85,B 0,C 180,E1 -22565.039,E2 -22565.039} C_VEL
LIN {X 0,Y 184.227,Z 747.578,A -85,B 0,C 180,E1 -22568.162,E2 -22568.162} C_VEL
LIN {X 0,Y 182.004,Z 752.822,A -85,B 0,C 180,E1 -22570.837,E2 -22570.837} C_VEL
LIN {X 0,Y 179.873,Z 757.903,A -85,B 0,C 180,E1 -22574.125,E2 -22574.125} C_VEL
LIN {X 0,Y 178.194,Z 761.844,A -85,B 0,C 180,E1 -22577.47,E2 -22577.47} C_VEL
LIN {X 0,Y 177.096,Z 764.75,A -85,B 0,C 180,E1 -22580.864,E2 -22580.864} C_VEL
LIN {X 0,Y 176.358,Z 766.998,A -85,B 0,C 180,E1 -22585.053,E2 -22585.053} C_VEL
LIN {X 0,Y 176.145,Z 767.735,A -85,B 0,C 180,E1 -22587.711,E2 -22587.711} C_VEL
LIN {X 0,Y 176.121,Z 767.962,A -85,B 0,C 180,E1 -22589.998,E2 -22589.998} C_VEL
LIN {X 0,Y 176.144,Z 767.768,A -85,B 0,C 180,E1 -22592.285,E2 -22592.285} C_VEL
LIN {X 0,Y 176.364,Z 767.046,A -85,B 0,C 180,E1 -22594.968,E2 -22594.968} C_VEL
LIN {X 0,Y 177.094,Z 764.863,A -85,B 0,C 180,E1 -22599.132,E2 -22599.132} C_VEL
LIN {X 0,Y 178.186,Z 761.993,A -85,B 0,C 180,E1 -22602.527,E2 -22602.527} C_VEL
LIN {X 0,Y 179.803,Z 758.099,A -85,B 0,C 180,E1 -22605.877,E2 -22605.877} C_VEL
LIN {X 0,Y 181.936,Z 753.078,A -85,B 0,C 180,E1 -22609.166,E2 -22609.166} C_VEL
LIN {X 0,Y 184.619,Z 746.751,A -85,B 0,C 180,E1 -22612.373,E2 -22612.373} C_VEL
LIN {X 0,Y 187.845,Z 738.829,A -85,B 0,C 180,E1 -22615.482,E2 -22615.482} C_VEL
LIN {X 0,Y 190.954,Z 730.052,A -85,B 0,C 180,E1 -22618.222,E2 -22618.222} C_VEL
LIN {X 0,Y 194.293,Z 719.803,A -85,B 0,C 180,E1 -22620.724,E2 -22620.724} C_VEL
LIN {X 0,Y 197.636,Z 708.383,A -85,B 0,C 180,E1 -22622.838,E2 -22622.838} C_VEL
LIN {X 0,Y 200.424,Z 697.152,A -85,B 0,C 180,E1 -22624.43,E2 -22624.43} C_VEL
LIN {X 0,Y 202.604,Z 685.731,A -85,B 0,C 180,E1 -22625.673,E2 -22625.673} C_VEL
LIN {X 0,Y 204.418,Z 672.715,A -85,B 0,C 180,E1 -22626.673,E2 -22626.673} C_VEL
LIN {X 0,Y 205.562,Z 660.437,A -85,B 0,C 180,E1 -22627.263,E2 -22627.263} C_VEL
LIN {X 0,Y 207.941,Z 614.058,A -85,B 0,C 180,E1 -22628.769,E2 -22628.769} C_VEL
LIN {X 0,Y 201.33,Z 598.589,A -85,B 0,C 180,E1 -22631.022,E2 -22631.022} C_VEL
LIN {X 0,Y 197.935,Z 592.053,A -85,B 0,C 180,E1 -22632.201,E2 -22632.201} C_VEL
LIN {X 0,Y 191.943,Z 582.436,A -85,B 0,C 180,E1 -22634.348,E2 -22634.348} C_VEL
LIN {X 0,Y 186.906,Z 575.04,A -85,B 0,C 180,E1 -22636.29,E2 -22636.29} C_VEL
LIN {X 0,Y 184.509,Z 571.566,A -85,B 0,C 180,E1 -22637.274,E2 -22637.274} C_VEL
LIN {X 0,Y 182.16,Z 568.282,A -85,B 0,C 180,E1 -22638.277,E2 -22638.277} C_VEL
LIN {X 0,Y 181.392,Z 567.165,A -85,B 0,C 180,E1 -22638.617,E2 -22638.617} C_VEL
LIN {X 0,Y 179.349,Z 564.874,A -85,B 0,C 180,E1 -22639.507,E2 -22639.507} C_VEL
LIN {X 0,Y 178.492,Z 562.218,A -85,B 0,C 180,E1 -22640.037,E2 -22640.037} C_VEL
LIN {X 0,Y 178.492,Z 562.251,A -85,B 0,C 180,E1 -22645.773,E2 -22645.773} C_VEL
LIN {X 0,Y 178.518,Z 562.249,A -85,B 0,C 180,E1 -22650.005,E2 -22650.005} C_VEL
LIN {X 0,Y 178.529,Z 562.247,A -85,B 0,C 180,E1 -22654.874,E2 -22654.874} C_VEL
LIN {X 0,Y 178.633,Z 562.233,A -85,B 0,C 180,E1 -22660.769,E2 -22660.769} C_VEL
LIN {X 0,Y 178.676,Z 562.226,A -85,B 0,C 180,E1 -22666.349,E2 -22666.349} C_VEL
LIN {X 0,Y 178.957,Z 562.173,A -85,B 0,C 180,E1 -22670.962,E2 -22670.962} C_VEL
LIN {X 0,Y 179.148,Z 562.149,A -85,B 0,C 180,E1 -22677.752,E2 -22677.752} C_VEL
LIN {X 0,Y 179.366,Z 562.143,A -85,B 0,C 180,E1 -22680,E2 -22680} C_VEL
LIN {X 0,Y 178.869,Z 562.185,A -85,B 0,C 180,E1 -22684.507,E2 -22684.507} C_VEL
LIN {X 0,Y 178.972,Z 562.174,A -85,B 0,C 180,E1 -22689.037,E2 -22689.037} C_VEL
LIN {X 0,Y 178.677,Z 562.227,A -85,B 0,C 180,E1 -22693.651,E2 -22693.651} C_VEL
LIN {X 0,Y 178.633,Z 562.235,A -85,B 0,C 180,E1 -22699.231,E2 -22699.231} C_VEL
LIN {X 0,Y 178.529,Z 562.242,A -85,B 0,C 180,E1 -22705.125,E2 -22705.125} C_VEL
LIN {X 0,Y 178.471,Z 562.244,A -85,B 0,C 180,E1 -22710.792,E2 -22710.792} C_VEL
LIN {X 0,Y 178.481,Z 562.236,A -85,B 0,C 180,E1 -22714.221,E2 -22714.221} C_VEL
LIN {X 0,Y 178.527,Z 562.374,A -85,B 0,C 180,E1 -22718.067,E2 -22718.067} C_VEL
LIN {X 0,Y 179.289,Z 564.934,A -85,B 0,C 180,E1 -22720.024,E2 -22720.024} C_VEL
LIN {X 0,Y 181.779,Z 569.11,A -85,B 0,C 180,E1 -22721.275,E2 -22721.275} C_VEL
LIN {X 0,Y 186.53,Z 576.551,A -85,B 0,C 180,E1 -22723.311,E2 -22723.311} C_VEL
LIN {X 0,Y 191.843,Z 585.725,A -85,B 0,C 180,E1 -22725.431,E2 -22725.431} C_VEL
LIN {X 0,Y 197.413,Z 596.57,A -85,B 0,C 180,E1 -22727.518,E2 -22727.518} C_VEL
LIN {X 0,Y 203.977,Z 611.568,A -85,B 0,C 180,E1 -22729.852,E2 -22729.852} C_VEL
LIN {X 0,Y 206.537,Z 618.72,A -85,B 0,C 180,E1 -22730.759,E2 -22730.759} C_VEL
LIN {X 0,Y 207.332,Z 627.391,A -85,B 0,C 180,E1 -22731.314,E2 -22731.314} C_VEL
LIN {X 0,Y 206.912,Z 635.218,A -85,B 0,C 180,E1 -22731.561,E2 -22731.561} C_VEL
LIN {X 0,Y 206.089,Z 641.065,A -85,B 0,C 180,E1 -22731.635,E2 -22731.635} C_VEL
LIN {X 0,Y 200.54,Z 660.071,A -85,B 0,C 180,E1 -22731.236,E2 -22731.236} C_VEL
LIN {X 0,Y 199.742,Z 665.916,A -85,B 0,C 180,E1 -22731.316,E2 -22731.316} C_VEL
LIN {X 0,Y 198.593,Z 679.71,A -85,B 0,C 180,E1 -22731.915,E2 -22731.915} C_VEL
LIN {X 0,Y 196.483,Z 693.346,A -85,B 0,C 180,E1 -22732.874,E2 -22732.874} C_VEL
LIN {X 0,Y 194.186,Z 704.302,A -85,B 0,C 180,E1 -22733.979,E2 -22733.979} C_VEL
LIN {X 0,Y 191.206,Z 716.088,A -85,B 0,C 180,E1 -22735.591,E2 -22735.591} C_VEL
LIN {X 0,Y 187.59,Z 727.849,A -85,B 0,C 180,E1 -22737.735,E2 -22737.735} C_VEL
LIN {X 0,Y 183.915,Z 738.297,A -85,B 0,C 180,E1 -22740.216,E2 -22740.216} C_VEL
LIN {X 0,Y 180.668,Z 746.757,A -85,B 0,C 180,E1 -22742.804,E2 -22742.804} C_VEL
LIN {X 0,Y 177.455,Z 754.977,A -85,B 0,C 180,E1 -22746.027,E2 -22746.027} C_VEL
LIN {X 0,Y 174.547,Z 761.687,A -85,B 0,C 180,E1 -22749.374,E2 -22749.374} C_VEL
LIN {X 0,Y 171.88,Z 767.781,A -85,B 0,C 180,E1 -22753.37,E2 -22753.37} C_VEL
LIN {X 0,Y 170.407,Z 771.754,A -85,B 0,C 180,E1 -22756.892,E2 -22756.892} C_VEL
LIN {X 0,Y 169.424,Z 774.692,A -85,B 0,C 180,E1 -22760.451,E2 -22760.451} C_VEL
LIN {X 0,Y 169.073,Z 776.09,A -85,B 0,C 180,E1 -22762.838,E2 -22762.838} C_VEL
LIN {X 0,Y 168.858,Z 777.698,A -85,B 0,C 180,E1 -22767.617,E2 -22767.617} C_VEL
LIN {X 0,Y 168.955,Z 777.913,A -85,B 0,C 180,E1 -22770.002,E2 -22770.002} C_VEL
LIN {X 0,Y 169.055,Z 777.689,A -85,B 0,C 180,E1 -22772.385,E2 -22772.385} C_VEL
LIN {X 0,Y 169.396,Z 776.893,A -85,B 0,C 180,E1 -22775.298,E2 -22775.298} C_VEL
LIN {X 0,Y 170.22,Z 775.4,A -85,B 0,C 180,E1 -22778.834,E2 -22778.834} C_VEL
LIN {X 0,Y 170.834,Z 778.208,A -85,B 0,C 180,E1 -22781.872,E2 -22781.872} C_VEL
LIN {X 0,Y 173.116,Z 781.333,A -85,B 0,C 180,E1 -22786.512,E2 -22786.512} C_VEL
LIN {X 0,Y 174.769,Z 782.176,A -85,B 0,C 180,E1 -22788.768,E2 -22788.768} C_VEL
LIN {X 0,Y 179.072,Z 782.687,A -85,B 0,C 180,E1 -22793.11,E2 -22793.11} C_VEL
LIN {X 0,Y 181.845,Z 782.337,A -85,B 0,C 180,E1 -22795.161,E2 -22795.161} C_VEL
LIN {X 0,Y 188.309,Z 780.235,A -85,B 0,C 180,E1 -22799.026,E2 -22799.026} C_VEL
LIN {X 0,Y 193.857,Z 777.552,A -85,B 0,C 180,E1 -22801.716,E2 -22801.716} C_VEL
LIN {X 0,Y 199.946,Z 773.778,A -85,B 0,C 180,E1 -22804.223,E2 -22804.223} C_VEL
LIN {X 0,Y 206.562,Z 768.913,A -85,B 0,C 180,E1 -22806.544,E2 -22806.544} C_VEL
LIN {X 0,Y 214.979,Z 761.393,A -85,B 0,C 180,E1 -22809.001,E2 -22809.001} C_VEL
LIN {X 0,Y 221.375,Z 754.663,A -85,B 0,C 180,E1 -22810.605,E2 -22810.605} C_VEL
LIN {X 0,Y 228.447,Z 746.053,A -85,B 0,C 180,E1 -22812.181,E2 -22812.181} C_VEL
LIN {X 0,Y 234.99,Z 736.546,A -85,B 0,C 180,E1 -22813.464,E2 -22813.464} C_VEL
LIN {X 0,Y 241.508,Z 725.158,A -85,B 0,C 180,E1 -22814.593,E2 -22814.593} C_VEL
LIN {X 0,Y 246.647,Z 713.994,A -85,B 0,C 180,E1 -22815.428,E2 -22815.428} C_VEL
LIN {X 0,Y 247.406,Z 712.065,A -85,B 0,C 180,E1 -22815.552,E2 -22815.552} C_VEL
LIN {X 0,Y 247.143,Z 712.826,A -85,B 0,C 180,E1 -22815.988,E2 -22815.988} C_VEL
LIN {X 0,Y 242.136,Z 724.358,A -85,B 0,C 180,E1 -22816.783,E2 -22816.783} C_VEL
LIN {X 0,Y 236.501,Z 734.645,A -85,B 0,C 180,E1 -22817.752,E2 -22817.752} C_VEL
LIN {X 0,Y 230.875,Z 743.267,A -85,B 0,C 180,E1 -22818.831,E2 -22818.831} C_VEL
LIN {X 0,Y 223.443,Z 752.875,A -85,B 0,C 180,E1 -22820.437,E2 -22820.437} C_VEL
LIN {X 0,Y 216.989,Z 759.842,A -85,B 0,C 180,E1 -22822.02,E2 -22822.02} C_VEL
LIN {X 0,Y 209.627,Z 766.688,A -85,B 0,C 180,E1 -22824.076,E2 -22824.076} C_VEL
LIN {X 0,Y 202.526,Z 772.066,A -85,B 0,C 180,E1 -22826.394,E2 -22826.394} C_VEL
LIN {X 0,Y 196.393,Z 775.865,A -85,B 0,C 180,E1 -22828.742,E2 -22828.742} C_VEL
LIN {X 0,Y 190.574,Z 778.662,A -85,B 0,C 180,E1 -22831.353,E2 -22831.353} C_VEL
LIN {X 0,Y 187.054,Z 779.974,A -85,B 0,C 180,E1 -22833.201,E2 -22833.201} C_VEL
LIN {X 0,Y 183.851,Z 780.837,A -85,B 0,C 180,E1 -22835.134,E2 -22835.134} C_VEL
LIN {X 0,Y 178.265,Z 781.084,A -85,B 0,C 180,E1 -22839.218,E2 -22839.218} C_VEL
LIN {X 0,Y 176.041,Z 780.636,A -85,B 0,C 180,E1 -22841.375,E2 -22841.375} C_VEL
LIN {X 0,Y 174.153,Z 779.688,A -85,B 0,C 180,E1 -22843.591,E2 -22843.591} C_VEL
LIN {X 0,Y 172.649,Z 778.281,A -85,B 0,C 180,E1 -22845.863,E2 -22845.863} C_VEL
LIN {X 0,Y 171.089,Z 775.379,A -85,B 0,C 180,E1 -22849.348,E2 -22849.348} C_VEL
LIN {X 0,Y 170.2,Z 771.419,A -85,B 0,C 180,E1 -22852.884,E2 -22852.884} C_VEL
LIN {X 0,Y 170.151,Z 766.183,A -85,B 0,C 180,E1 -22856.448,E2 -22856.448} C_VEL
LIN {X 0,Y 170.429,Z 759.307,A -85,B 0,C 180,E1 -22860,E2 -22860} C_VEL
LIN {X 0,Y 170.71,Z 753.691,A -85,B 0,C 180,E1 -22862.36,E2 -22862.36} C_VEL
LIN {X 0,Y 170.987,Z 746.81,A -85,B 0,C 180,E1 -22864.715,E2 -22864.715} C_VEL
LIN {X 0,Y 171.355,Z 737.345,A -85,B 0,C 180,E1 -22867.364,E2 -22867.364} C_VEL
LIN {X 0,Y 171.936,Z 726.978,A -85,B 0,C 180,E1 -22869.624,E2 -22869.624} C_VEL
LIN {X 0,Y 172.48,Z 716.295,A -85,B 0,C 180,E1 -22871.466,E2 -22871.466} C_VEL
LIN {X 0,Y 172.946,Z 704.161,A -85,B 0,C 180,E1 -22873.012,E2 -22873.012} C_VEL
LIN {X 0,Y 173.364,Z 688.853,A -85,B 0,C 180,E1 -22874.377,E2 -22874.377} C_VEL
LIN {X 0,Y 174.238,Z 645.682,A -85,B 0,C 180,E1 -22877.723,E2 -22877.723} C_VEL
LIN {X 0,Y 172.719,Z 622.516,A -85,B 0,C 180,E1 -22879.445,E2 -22879.445} C_VEL
LIN {X 0,Y 172.648,Z 617.452,A -85,B 0,C 180,E1 -22879.901,E2 -22879.901} C_VEL
LIN {X 0,Y 175.171,Z 593.393,A -85,B 0,C 180,E1 -22887.379,E2 -22887.379} C_VEL
LIN {X 0,Y 176.067,Z 585.107,A -85,B 0,C 180,E1 -22889.931,E2 -22889.931} C_VEL
LIN {X 0,Y 172.585,Z 568.074,A -85,B 0,C 180,E1 -22895.465,E2 -22895.465} C_VEL
LIN {X 0,Y 171.866,Z 564.602,A -85,B 0,C 180,E1 -22896.735,E2 -22896.735} C_VEL
LIN {X 0,Y 171.776,Z 564.148,A -85,B 0,C 180,E1 -22897.227,E2 -22897.227} C_VEL
LIN {X 0,Y 171.947,Z 564.767,A -85,B 0,C 180,E1 -22897.656,E2 -22897.656} C_VEL
LIN {X 0,Y 173.601,Z 567.383,A -85,B 0,C 180,E1 -22898.59,E2 -22898.59} C_VEL
LIN {X 0,Y 175.041,Z 568.614,A -85,B 0,C 180,E1 -22899.261,E2 -22899.261} C_VEL
LIN {X 0,Y 177.197,Z 572.04,A -85,B 0,C 180,E1 -22900.324,E2 -22900.324} C_VEL
LIN {X 0,Y 178.786,Z 573.978,A -85,B 0,C 180,E1 -22901.042,E2 -22901.042} C_VEL
LIN {X 0,Y 184.709,Z 582.522,A -85,B 0,C 180,E1 -22903.602,E2 -22903.602} C_VEL
LIN {X 0,Y 191.145,Z 592.516,A -85,B 0,C 180,E1 -22906.121,E2 -22906.121} C_VEL
LIN {X 0,Y 195.424,Z 600.18,A -85,B 0,C 180,E1 -22907.701,E2 -22907.701} C_VEL
LIN {X 0,Y 200.817,Z 612.479,A -85,B 0,C 180,E1 -22909.666,E2 -22909.666} C_VEL
LIN {X 0,Y 202.208,Z 615.933,A -85,B 0,C 180,E1 -22910.16,E2 -22910.16} C_VEL
LIN {X 0,Y 199.5,Z 664.831,A -85,B 0,C 180,E1 -22911.809,E2 -22911.809} C_VEL
LIN {X 0,Y 197.95,Z 678.229,A -85,B 0,C 180,E1 -22912.612,E2 -22912.612} C_VEL
LIN {X 0,Y 195.901,Z 690.378,A -85,B 0,C 180,E1 -22913.703,E2 -22913.703} C_VEL
LIN {X 0,Y 193.437,Z 701.658,A -85,B 0,C 180,E1 -22915.092,E2 -22915.092} C_VEL
LIN {X 0,Y 190.211,Z 713.286,A -85,B 0,C 180,E1 -22916.974,E2 -22916.974} C_VEL
LIN {X 0,Y 186.902,Z 723.728,A -85,B 0,C 180,E1 -22919.179,E2 -22919.179} C_VEL
LIN {X 0,Y 183.624,Z 732.997,A -85,B 0,C 180,E1 -22921.679,E2 -22921.679} C_VEL
LIN {X 0,Y 180.346,Z 741.493,A -85,B 0,C 180,E1 -22924.615,E2 -22924.615} C_VEL
LIN {X 0,Y 177.144,Z 748.895,A -85,B 0,C 180,E1 -22927.856,E2 -22927.856} C_VEL
LIN {X 0,Y 174.495,Z 754.835,A -85,B 0,C 180,E1 -22931.201,E2 -22931.201} C_VEL
LIN {X 0,Y 172.377,Z 759.525,A -85,B 0,C 180,E1 -22934.63,E2 -22934.63} C_VEL
LIN {X 0,Y 170.821,Z 763.107,A -85,B 0,C 180,E1 -22938.127,E2 -22938.127} C_VEL
LIN {X 0,Y 170.1,Z 764.955,A -85,B 0,C 180,E1 -22940.485,E2 -22940.485} C_VEL
LIN {X 0,Y 169.586,Z 766.343,A -85,B 0,C 180,E1 -22942.856,E2 -22942.856} C_VEL
LIN {X 0,Y 169.258,Z 767.332,A -85,B 0,C 180,E1 -22945.234,E2 -22945.234} C_VEL
LIN {X 0,Y 169.063,Z 767.939,A -85,B 0,C 180,E1 -22947.615,E2 -22947.615} C_VEL
LIN {X 0,Y 169.033,Z 768.166,A -85,B 0,C 180,E1 -22949.998,E2 -22949.998} C_VEL
LIN {X 0,Y 169.062,Z 767.973,A -85,B 0,C 180,E1 -22952.38,E2 -22952.38} C_VEL
LIN {X 0,Y 169.257,Z 767.388,A -85,B 0,C 180,E1 -22954.762,E2 -22954.762} C_VEL
LIN {X 0,Y 170.098,Z 765.067,A -85,B 0,C 180,E1 -22959.511,E2 -22959.511} C_VEL
LIN {X 0,Y 171.267,Z 762.197,A -85,B 0,C 180,E1 -22963.042,E2 -22963.042} C_VEL
LIN {X 0,Y 172.978,Z 758.303,A -85,B 0,C 180,E1 -22966.521,E2 -22966.521} C_VEL
LIN {X 0,Y 175.234,Z 753.282,A -85,B 0,C 180,E1 -22969.93,E2 -22969.93} C_VEL
LIN {X 0,Y 178.073,Z 746.953,A -85,B 0,C 180,E1 -22973.243,E2 -22973.243} C_VEL
LIN {X 0,Y 181.455,Z 739.031,A -85,B 0,C 180,E1 -22976.447,E2 -22976.447} C_VEL
LIN {X 0,Y 184.474,Z 730.922,A -85,B 0,C 180,E1 -22979.072,E2 -22979.072} C_VEL
LIN {X 0,Y 187.883,Z 721.106,A -85,B 0,C 180,E1 -22981.578,E2 -22981.578} C_VEL
LIN {X 0,Y 191.331,Z 710.004,A -85,B 0,C 180,E1 -22983.748,E2 -22983.748} C_VEL
LIN {X 0,Y 194.193,Z 699.114,A -85,B 0,C 180,E1 -22985.381,E2 -22985.381} C_VEL
LIN {X 0,Y 196.682,Z 687.068,A -85,B 0,C 180,E1 -22986.762,E2 -22986.762} C_VEL
LIN {X 0,Y 198.651,Z 674.06,A -85,B 0,C 180,E1 -22987.82,E2 -22987.82} C_VEL
LIN {X 0,Y 199.938,Z 661.056,A -85,B 0,C 180,E1 -22988.476,E2 -22988.476} C_VEL
LIN {X 0,Y 202.355,Z 616.192,A -85,B 0,C 180,E1 -22989.962,E2 -22989.962} C_VEL
LIN {X 0,Y 196.641,Z 602.592,A -85,B 0,C 180,E1 -22992.035,E2 -22992.035} C_VEL
LIN {X 0,Y 193.03,Z 595.589,A -85,B 0,C 180,E1 -22993.366,E2 -22993.366} C_VEL
LIN {X 0,Y 186.369,Z 584.942,A -85,B 0,C 180,E1 -22995.922,E2 -22995.922} C_VEL
LIN {X 0,Y 180.925,Z 576.999,A -85,B 0,C 180,E1 -22998.207,E2 -22998.207} C_VEL
LIN {X 0,Y 177.806,Z 572.682,A -85,B 0,C 180,E1 -22999.615,E2 -22999.615} C_VEL
LIN {X 0,Y 175.574,Z 569.643,A -85,B 0,C 180,E1 -23000.677,E2 -23000.677} C_VEL
LIN {X 0,Y 174.742,Z 568.282,A -85,B 0,C 180,E1 -23001.101,E2 -23001.101} C_VEL
LIN {X 0,Y 172.531,Z 566.133,A -85,B 0,C 180,E1 -23002.17,E2 -23002.17} C_VEL
LIN {X 0,Y 171.473,Z 563.585,A -85,B 0,C 180,E1 -23002.804,E2 -23002.804} C_VEL
LIN {X 0,Y 171.403,Z 563.102,A -85,B 0,C 180,E1 -23002.97,E2 -23002.97} C_VEL
LIN {X 0,Y 171.423,Z 563.12,A -85,B 0,C 180,E1 -23007.793,E2 -23007.793} C_VEL
LIN {X 0,Y 171.444,Z 563.125,A -85,B 0,C 180,E1 -23010.533,E2 -23010.533} C_VEL
LIN {X 0,Y 171.453,Z 563.123,A -85,B 0,C 180,E1 -23015.801,E2 -23015.801} C_VEL
LIN {X 0,Y 171.59,Z 563.11,A -85,B 0,C 180,E1 -23020.873,E2 -23020.873} C_VEL
LIN {X 0,Y 171.591,Z 563.102,A -85,B 0,C 180,E1 -23025.774,E2 -23025.774} C_VEL
LIN {X 0,Y 171.885,Z 563.052,A -85,B 0,C 180,E1 -23030.587,E2 -23030.587} C_VEL
LIN {X 0,Y 171.818,Z 563.068,A -85,B 0,C 180,E1 -23035.307,E2 -23035.307} C_VEL
LIN {X 0,Y 172.329,Z 563.02,A -85,B 0,C 180,E1 -23040,E2 -23040} C_VEL
LIN {X 0,Y 171.819,Z 563.064,A -85,B 0,C 180,E1 -23044.692,E2 -23044.692} C_VEL
LIN {X 0,Y 171.904,Z 563.052,A -85,B 0,C 180,E1 -23049.412,E2 -23049.412} C_VEL
LIN {X 0,Y 171.592,Z 563.104,A -85,B 0,C 180,E1 -23054.226,E2 -23054.226} C_VEL
LIN {X 0,Y 171.552,Z 563.114,A -85,B 0,C 180,E1 -23059.575,E2 -23059.575} C_VEL
LIN {X 0,Y 171.463,Z 563.118,A -85,B 0,C 180,E1 -23065.617,E2 -23065.617} C_VEL
LIN {X 0,Y 171.434,Z 563.121,A -85,B 0,C 180,E1 -23070.587,E2 -23070.587} C_VEL
LIN {X 0,Y 171.402,Z 563.184,A -85,B 0,C 180,E1 -23075.753,E2 -23075.753} C_VEL
LIN {X 0,Y 171.725,Z 564.407,A -85,B 0,C 180,E1 -23076.857,E2 -23076.857} C_VEL
LIN {X 0,Y 174.542,Z 568.945,A -85,B 0,C 180,E1 -23078.499,E2 -23078.499} C_VEL
LIN {X 0,Y 176.125,Z 571.158,A -85,B 0,C 180,E1 -23079.277,E2 -23079.277} C_VEL
LIN {X 0,Y 179.948,Z 577.158,A -85,B 0,C 180,E1 -23081.09,E2 -23081.09} C_VEL
LIN {X 0,Y 183.331,Z 582.76,A -85,B 0,C 180,E1 -23082.598,E2 -23082.598} C_VEL
LIN {X 0,Y 187.994,Z 591.096,A -85,B 0,C 180,E1 -23084.558,E2 -23084.558} C_VEL
LIN {X 0,Y 192.985,Z 600.997,A -85,B 0,C 180,E1 -23086.532,E2 -23086.532} C_VEL
LIN {X 0,Y 198.68,Z 614.322,A -85,B 0,C 180,E1 -23088.689,E2 -23088.689} C_VEL
LIN {X 0,Y 201.096,Z 620.643,A -85,B 0,C 180,E1 -23089.578,E2 -23089.578} C_VEL
LIN {X 0,Y 201.761,Z 628.427,A -85,B 0,C 180,E1 -23090.091,E2 -23090.091} C_VEL
LIN {X 0,Y 199.742,Z 665.916,A -85,B 0,C 180,E1 -23091.316,E2 -23091.316} C_VEL
LIN {X 0,Y 198.879,Z 671.754,A -85,B 0,C 180,E1 -23091.417,E2 -23091.417} C_VEL
LIN {X 0,Y 195.689,Z 681.156,A -85,B 0,C 180,E1 -23091.371,E2 -23091.371} C_VEL
LIN {X 0,Y 191.981,Z 690.373,A -85,B 0,C 180,E1 -23091.476,E2 -23091.476} C_VEL
LIN {X 0,Y 190.313,Z 695.925,A -85,B 0,C 180,E1 -23091.838,E2 -23091.838} C_VEL
LIN {X 0,Y 187.611,Z 707.766,A -85,B 0,C 180,E1 -23093.178,E2 -23093.178} C_VEL
LIN {X 0,Y 184.543,Z 718.744,A -85,B 0,C 180,E1 -23094.832,E2 -23094.832} C_VEL
LIN {X 0,Y 180.815,Z 729.946,A -85,B 0,C 180,E1 -23097.035,E2 -23097.035} C_VEL
LIN {X 0,Y 177.05,Z 739.888,A -85,B 0,C 180,E1 -23099.597,E2 -23099.597} C_VEL
LIN {X 0,Y 173.751,Z 748.046,A -85,B 0,C 180,E1 -23102.282,E2 -23102.282} C_VEL
LIN {X 0,Y 170.407,Z 756.06,A -85,B 0,C 180,E1 -23105.645,E2 -23105.645} C_VEL
LIN {X 0,Y 167.483,Z 762.478,A -85,B 0,C 180,E1 -23109.106,E2 -23109.106} C_VEL
LIN {X 0,Y 165.071,Z 767.576,A -85,B 0,C 180,E1 -23112.663,E2 -23112.663} C_VEL
LIN {X 0,Y 163.457,Z 771.549,A -85,B 0,C 180,E1 -23116.324,E2 -23116.324} C_VEL
LIN {X 0,Y 162.404,Z 774.488,A -85,B 0,C 180,E1 -23120.034,E2 -23120.034} C_VEL
LIN {X 0,Y 161.999,Z 775.885,A -85,B 0,C 180,E1 -23122.524,E2 -23122.524} C_VEL
LIN {X 0,Y 161.791,Z 776.884,A -85,B 0,C 180,E1 -23125.018,E2 -23125.018} C_VEL
LIN {X 0,Y 161.764,Z 777.548,A -85,B 0,C 180,E1 -23127.792,E2 -23127.792} C_VEL
LIN {X 0,Y 161.855,Z 777.708,A -85,B 0,C 180,E1 -23130.002,E2 -23130.002} C_VEL
LIN {X 0,Y 161.974,Z 777.485,A -85,B 0,C 180,E1 -23132.489,E2 -23132.489} C_VEL
LIN {X 0,Y 162.255,Z 776.871,A -85,B 0,C 180,E1 -23134.972,E2 -23134.972} C_VEL
LIN {X 0,Y 163.52,Z 774.623,A -85,B 0,C 180,E1 -23139.98,E2 -23139.98} C_VEL
LIN {X 0,Y 165.021,Z 778.935,A -85,B 0,C 180,E1 -23144.807,E2 -23144.807} C_VEL
LIN {X 0,Y 168.103,Z 781.549,A -85,B 0,C 180,E1 -23149.542,E2 -23149.542} C_VEL
LIN {X 0,Y 170.111,Z 782.328,A -85,B 0,C 180,E1 -23151.83,E2 -23151.83} C_VEL
LIN {X 0,Y 172.576,Z 782.593,A -85,B 0,C 180,E1 -23154.034,E2 -23154.034} C_VEL
LIN {X 0,Y 178.653,Z 782.027,A -85,B 0,C 180,E1 -23158.17,E2 -23158.17} C_VEL
LIN {X 0,Y 182.175,Z 781.088,A -85,B 0,C 180,E1 -23160.102,E2 -23160.102} C_VEL
LIN {X 0,Y 189.996,Z 777.902,A -85,B 0,C 180,E1 -23163.703,E2 -23163.703} C_VEL
LIN {X 0,Y 196.493,Z 774.337,A -85,B 0,C 180,E1 -23166.17,E2 -23166.17} C_VEL
LIN {X 0,Y 203.529,Z 769.623,A -85,B 0,C 180,E1 -23168.431,E2 -23168.431} C_VEL
LIN {X 0,Y 211.105,Z 763.633,A -85,B 0,C 180,E1 -23170.482,E2 -23170.482} C_VEL
LIN {X 0,Y 219.108,Z 756.035,A -85,B 0,C 180,E1 -23172.346,E2 -23172.346} C_VEL
LIN {X 0,Y 225.788,Z 748.537,A -85,B 0,C 180,E1 -23173.722,E2 -23173.722} C_VEL
LIN {X 0,Y 233.323,Z 738.759,A -85,B 0,C 180,E1 -23175.062,E2 -23175.062} C_VEL
LIN {X 0,Y 236.318,Z 734.163,A -85,B 0,C 180,E1 -23175.542,E2 -23175.542} C_VEL
LIN {X 0,Y 235.558,Z 735.394,A -85,B 0,C 180,E1 -23176.018,E2 -23176.018} C_VEL
LIN {X 0,Y 229.166,Z 744.673,A -85,B 0,C 180,E1 -23177.144,E2 -23177.144} C_VEL
LIN {X 0,Y 222.474,Z 752.746,A -85,B 0,C 180,E1 -23178.441,E2 -23178.441} C_VEL
LIN {X 0,Y 215.666,Z 759.71,A -85,B 0,C 180,E1 -23179.939,E2 -23179.939} C_VEL
LIN {X 0,Y 209.13,Z 765.512,A -85,B 0,C 180,E1 -23181.559,E2 -23181.559} C_VEL
LIN {X 0,Y 201.697,Z 771.062,A -85,B 0,C 180,E1 -23183.676,E2 -23183.676} C_VEL
LIN {X 0,Y 195.893,Z 774.672,A -85,B 0,C 180,E1 -23185.608,E2 -23185.608} C_VEL
LIN {X 0,Y 188.382,Z 778.258,A -85,B 0,C 180,E1 -23188.513,E2 -23188.513} C_VEL
LIN {X 0,Y 184.447,Z 779.734,A -85,B 0,C 180,E1 -23190.308,E2 -23190.308} C_VEL
LIN {X 0,Y 180.789,Z 780.644,A -85,B 0,C 180,E1 -23192.193,E2 -23192.193} C_VEL
LIN {X 0,Y 174.448,Z 781.299,A -85,B 0,C 180,E1 -23196.242,E2 -23196.242} C_VEL
LIN {X 0,Y 171.671,Z 780.95,A -85,B 0,C 180,E1 -23198.38,E2 -23198.38} C_VEL
LIN {X 0,Y 167.415,Z 778.962,A -85,B 0,C 180,E1 -23202.911,E2 -23202.911} C_VEL
LIN {X 0,Y 165.218,Z 776.349,A -85,B 0,C 180,E1 -23206.47,E2 -23206.47} C_VEL
LIN {X 0,Y 163.955,Z 772.729,A -85,B 0,C 180,E1 -23210.127,E2 -23210.127} C_VEL
LIN {X 0,Y 163.34,Z 767.942,A -85,B 0,C 180,E1 -23213.825,E2 -23213.825} C_VEL
LIN {X 0,Y 163.398,Z 761.866,A -85,B 0,C 180,E1 -23217.535,E2 -23217.535} C_VEL
LIN {X 0,Y 163.77,Z 755.318,A -85,B 0,C 180,E1 -23220.615,E2 -23220.615} C_VEL
LIN {X 0,Y 164.045,Z 748.917,A -85,B 0,C 180,E1 -23223.07,E2 -23223.07} C_VEL
LIN {X 0,Y 164.386,Z 740.09,A -85,B 0,C 180,E1 -23225.828,E2 -23225.828} C_VEL
LIN {X 0,Y 164.805,Z 730.306,A -85,B 0,C 180,E1 -23228.275,E2 -23228.275} C_VEL
LIN {X 0,Y 165.389,Z 719.042,A -85,B 0,C 180,E1 -23230.423,E2 -23230.423} C_VEL
LIN {X 0,Y 165.874,Z 707.886,A -85,B 0,C 180,E1 -23232.068,E2 -23232.068} C_VEL
LIN {X 0,Y 166.188,Z 693.681,A -85,B 0,C 180,E1 -23233.51,E2 -23233.51} C_VEL
LIN {X 0,Y 167.272,Z 646.699,A -85,B 0,C 180,E1 -23237.419,E2 -23237.419} C_VEL
LIN {X 0,Y 165.658,Z 622.712,A -85,B 0,C 180,E1 -23239.276,E2 -23239.276} C_VEL
LIN {X 0,Y 165.54,Z 617.716,A -85,B 0,C 180,E1 -23239.694,E2 -23239.694} C_VEL
LIN {X 0,Y 168.031,Z 593.814,A -85,B 0,C 180,E1 -23247.393,E2 -23247.393} C_VEL
LIN {X 0,Y 168.995,Z 585.835,A -85,B 0,C 180,E1 -23249.937,E2 -23249.937} C_VEL
LIN {X 0,Y 166.2,Z 572.14,A -85,B 0,C 180,E1 -23254.627,E2 -23254.627} C_VEL
LIN {X 0,Y 166.201,Z 571.62,A -85,B 0,C 180,E1 -23255.37,E2 -23255.37} C_VEL
LIN {X 0,Y 167.145,Z 572.381,A -85,B 0,C 180,E1 -23256.062,E2 -23256.062} C_VEL
LIN {X 0,Y 169.885,Z 572.4,A -85,B 0,C 180,E1 -23257.324,E2 -23257.324} C_VEL
LIN {X 0,Y 172.111,Z 574.976,A -85,B 0,C 180,E1 -23258.463,E2 -23258.463} C_VEL
LIN {X 0,Y 174.877,Z 578.718,A -85,B 0,C 180,E1 -23259.836,E2 -23259.836} C_VEL
LIN {X 0,Y 181.769,Z 588.99,A -85,B 0,C 180,E1 -23262.982,E2 -23262.982} C_VEL
LIN {X 0,Y 187.476,Z 598.162,A -85,B 0,C 180,E1 -23265.324,E2 -23265.324} C_VEL
LIN {X 0,Y 191.047,Z 604.679,A -85,B 0,C 180,E1 -23266.714,E2 -23266.714} C_VEL
LIN {X 0,Y 196.17,Z 616.691,A -85,B 0,C 180,E1 -23268.696,E2 -23268.696} C_VEL
LIN {X 0,Y 196.698,Z 617.997,A -85,B 0,C 180,E1 -23268.894,E2 -23268.894} C_VEL
LIN {X 0,Y 193.94,Z 665.437,A -85,B 0,C 180,E1 -23270.533,E2 -23270.533} C_VEL
LIN {X 0,Y 192.295,Z 679.047,A -85,B 0,C 180,E1 -23271.379,E2 -23271.379} C_VEL
LIN {X 0,Y 190.022,Z 691.67,A -85,B 0,C 180,E1 -23272.557,E2 -23272.557} C_VEL
LIN {X 0,Y 187.197,Z 703.451,A -85,B 0,C 180,E1 -23274.081,E2 -23274.081} C_VEL
LIN {X 0,Y 183.941,Z 714.781,A -85,B 0,C 180,E1 -23276.026,E2 -23276.026} C_VEL
LIN {X 0,Y 180.464,Z 724.992,A -85,B 0,C 180,E1 -23278.28,E2 -23278.28} C_VEL
LIN {X 0,Y 176.774,Z 734.764,A -85,B 0,C 180,E1 -23281.1,E2 -23281.1} C_VEL
LIN {X 0,Y 173.383,Z 743.047,A -85,B 0,C 180,E1 -23284.165,E2 -23284.165} C_VEL
LIN {X 0,Y 170.075,Z 750.212,A -85,B 0,C 180,E1 -23287.526,E2 -23287.526} C_VEL
LIN {X 0,Y 167.77,Z 755.041,A -85,B 0,C 180,E1 -23290.418,E2 -23290.418} C_VEL
LIN {X 0,Y 165.539,Z 759.731,A -85,B 0,C 180,E1 -23293.979,E2 -23293.979} C_VEL
LIN {X 0,Y 163.877,Z 763.312,A -85,B 0,C 180,E1 -23297.616,E2 -23297.616} C_VEL
LIN {X 0,Y 163.087,Z 765.161,A -85,B 0,C 180,E1 -23300.072,E2 -23300.072} C_VEL
LIN {X 0,Y 162.548,Z 766.549,A -85,B 0,C 180,E1 -23302.545,E2 -23302.545} C_VEL
LIN {X 0,Y 162.126,Z 767.715,A -85,B 0,C 180,E1 -23305.586,E2 -23305.586} C_VEL
LIN {X 0,Y 161.946,Z 768.371,A -85,B 0,C 180,E1 -23309.998,E2 -23309.998} C_VEL
LIN {X 0,Y 162.099,Z 767.81,A -85,B 0,C 180,E1 -23314.288,E2 -23314.288} C_VEL
LIN {X 0,Y 162.547,Z 766.627,A -85,B 0,C 180,E1 -23317.451,E2 -23317.451} C_VEL
LIN {X 0,Y 163.084,Z 765.271,A -85,B 0,C 180,E1 -23319.924,E2 -23319.924} C_VEL
LIN {X 0,Y 164.341,Z 762.401,A -85,B 0,C 180,E1 -23323.601,E2 -23323.601} C_VEL
LIN {X 0,Y 166.183,Z 758.506,A -85,B 0,C 180,E1 -23327.217,E2 -23327.217} C_VEL
LIN {X 0,Y 168.571,Z 753.485,A -85,B 0,C 180,E1 -23330.753,E2 -23330.753} C_VEL
LIN {X 0,Y 171.575,Z 747.156,A -85,B 0,C 180,E1 -23334.178,E2 -23334.178} C_VEL
LIN {X 0,Y 175.116,Z 739.234,A -85,B 0,C 180,E1 -23337.484,E2 -23337.484} C_VEL
LIN {X 0,Y 178.21,Z 731.341,A -85,B 0,C 180,E1 -23340.119,E2 -23340.119} C_VEL
LIN {X 0,Y 181.872,Z 721.307,A -85,B 0,C 180,E1 -23342.749,E2 -23342.749} C_VEL
LIN {X 0,Y 185.485,Z 710.204,A -85,B 0,C 180,E1 -23344.963,E2 -23344.963} C_VEL
LIN {X 0,Y 188.461,Z 699.313,A -85,B 0,C 180,E1 -23346.629,E2 -23346.629} C_VEL
LIN {X 0,Y 191.062,Z 687.265,A -85,B 0,C 180,E1 -23348.031,E2 -23348.031} C_VEL
LIN {X 0,Y 193.036,Z 674.74,A -85,B 0,C 180,E1 -23349.081,E2 -23349.081} C_VEL
LIN {X 0,Y 194.411,Z 661.783,A -85,B 0,C 180,E1 -23349.752,E2 -23349.752} C_VEL
LIN {X 0,Y 196.865,Z 618.296,A -85,B 0,C 180,E1 -23351.223,E2 -23351.223} C_VEL
LIN {X 0,Y 191.177,Z 604.752,A -85,B 0,C 180,E1 -23353.429,E2 -23353.429} C_VEL
LIN {X 0,Y 186.151,Z 595.82,A -85,B 0,C 180,E1 -23355.401,E2 -23355.401} C_VEL
LIN {X 0,Y 179.776,Z 585.888,A -85,B 0,C 180,E1 -23358.096,E2 -23358.096} C_VEL
LIN {X 0,Y 176.654,Z 581.436,A -85,B 0,C 180,E1 -23359.518,E2 -23359.518} C_VEL
LIN {X 0,Y 174.195,Z 577.953,A -85,B 0,C 180,E1 -23360.703,E2 -23360.703} C_VEL
LIN {X 0,Y 171.391,Z 574.007,A -85,B 0,C 180,E1 -23362.135,E2 -23362.135} C_VEL
LIN {X 0,Y 168.911,Z 570.965,A -85,B 0,C 180,E1 -23363.451,E2 -23363.451} C_VEL
LIN {X 0,Y 168.035,Z 569.358,A -85,B 0,C 180,E1 -23363.973,E2 -23363.973} C_VEL
LIN {X 0,Y 165.777,Z 567.468,A -85,B 0,C 180,E1 -23365.209,E2 -23365.209} C_VEL
LIN {X 0,Y 164.503,Z 564.904,A -85,B 0,C 180,E1 -23366.054,E2 -23366.054} C_VEL
LIN {X 0,Y 164.328,Z 564.01,A -85,B 0,C 180,E1 -23366.221,E2 -23366.221} C_VEL
LIN {X 0,Y 164.401,Z 564.002,A -85,B 0,C 180,E1 -23369.136,E2 -23369.136} C_VEL
LIN {X 0,Y 164.411,Z 564.005,A -85,B 0,C 180,E1 -23374.693,E2 -23374.693} C_VEL
LIN {X 0,Y 164.48,Z 563.992,A -85,B 0,C 180,E1 -23380.049,E2 -23380.049} C_VEL
LIN {X 0,Y 164.535,Z 563.974,A -85,B 0,C 180,E1 -23385.15,E2 -23385.15} C_VEL
LIN {X 0,Y 164.799,Z 563.933,A -85,B 0,C 180,E1 -23390.178,E2 -23390.178} C_VEL
LIN {X 0,Y 164.849,Z 563.946,A -85,B 0,C 180,E1 -23392.652,E2 -23392.652} C_VEL
LIN {X 0,Y 165.044,Z 563.904,A -85,B 0,C 180,E1 -23397.559,E2 -23397.559} C_VEL
LIN {X 0,Y 165.291,Z 563.896,A -85,B 0,C 180,E1 -23400,E2 -23400} C_VEL
LIN {X 0,Y 164.856,Z 563.949,A -85,B 0,C 180,E1 -23407.348,E2 -23407.348} C_VEL
LIN {X 0,Y 164.774,Z 563.942,A -85,B 0,C 180,E1 -23411.198,E2 -23411.198} C_VEL
LIN {X 0,Y 164.493,Z 563.981,A -85,B 0,C 180,E1 -23417.402,E2 -23417.402} C_VEL
LIN {X 0,Y 164.469,Z 563.992,A -85,B 0,C 180,E1 -23419.99,E2 -23419.99} C_VEL
LIN {X 0,Y 164.387,Z 563.996,A -85,B 0,C 180,E1 -23426.134,E2 -23426.134} C_VEL
LIN {X 0,Y 164.373,Z 564.005,A -85,B 0,C 180,E1 -23432.375,E2 -23432.375} C_VEL
LIN {X 0,Y 164.347,Z 564.224,A -85,B 0,C 180,E1 -23433.336,E2 -23433.336} C_VEL
LIN {X 0,Y 165.468,Z 567.043,A -85,B 0,C 180,E1 -23434.244,E2 -23434.244} C_VEL
LIN {X 0,Y 168.685,Z 570.478,A -85,B 0,C 180,E1 -23436.05,E2 -23436.05} C_VEL
LIN {X 0,Y 173.024,Z 577.122,A -85,B 0,C 180,E1 -23438.403,E2 -23438.403} C_VEL
LIN {X 0,Y 176.766,Z 583.119,A -85,B 0,C 180,E1 -23440.268,E2 -23440.268} C_VEL
LIN {X 0,Y 181.077,Z 590.397,A -85,B 0,C 180,E1 -23442.264,E2 -23442.264} C_VEL
LIN {X 0,Y 187.182,Z 602.277,A -85,B 0,C 180,E1 -23444.903,E2 -23444.903} C_VEL
LIN {X 0,Y 193.333,Z 616.595,A -85,B 0,C 180,E1 -23447.402,E2 -23447.402} C_VEL
LIN {X 0,Y 195.875,Z 623.433,A -85,B 0,C 180,E1 -23448.407,E2 -23448.407} C_VEL
LIN {X 0,Y 196.319,Z 629.046,A -85,B 0,C 180,E1 -23448.788,E2 -23448.788} C_VEL
LIN {X 0,Y 193.665,Z 673.582,A -85,B 0,C 180,E1 -23450.304,E2 -23450.304} C_VEL
LIN {X 0,Y 191.97,Z 687.089,A -85,B 0,C 180,E1 -23451.109,E2 -23451.109} C_VEL
LIN {X 0,Y 190.313,Z 695.925,A -85,B 0,C 180,E1 -23451.838,E2 -23451.838} C_VEL
LIN {X 0,Y 188.509,Z 701.534,A -85,B 0,C 180,E1 -23452.28,E2 -23452.28} C_VEL
LIN {X 0,Y 183.954,Z 710.26,A -85,B 0,C 180,E1 -23452.83,E2 -23452.83} C_VEL
LIN {X 0,Y 179.242,Z 718.494,A -85,B 0,C 180,E1 -23453.611,E2 -23453.611} C_VEL
LIN {X 0,Y 177.203,Z 723.31,A -85,B 0,C 180,E1 -23454.405,E2 -23454.405} C_VEL
LIN {X 0,Y 173.267,Z 733.993,A -85,B 0,C 180,E1 -23456.801,E2 -23456.801} C_VEL
LIN {X 0,Y 169.497,Z 743.141,A -85,B 0,C 180,E1 -23459.477,E2 -23459.477} C_VEL
LIN {X 0,Y 165.689,Z 751.939,A -85,B 0,C 180,E1 -23462.812,E2 -23462.812} C_VEL
LIN {X 0,Y 162.283,Z 759.246,A -85,B 0,C 180,E1 -23466.387,E2 -23466.387} C_VEL
LIN {X 0,Y 159.074,Z 765.784,A -85,B 0,C 180,E1 -23470.651,E2 -23470.651} C_VEL
LIN {X 0,Y 157.008,Z 770.118,A -85,B 0,C 180,E1 -23474.423,E2 -23474.423} C_VEL
LIN {X 0,Y 156.086,Z 772.42,A -85,B 0,C 180,E1 -23476.992,E2 -23476.992} C_VEL
LIN {X 0,Y 155.405,Z 774.283,A -85,B 0,C 180,E1 -23479.58,E2 -23479.58} C_VEL
LIN {X 0,Y 154.949,Z 775.68,A -85,B 0,C 180,E1 -23482.182,E2 -23482.182} C_VEL
LIN {X 0,Y 154.711,Z 776.679,A -85,B 0,C 180,E1 -23484.79,E2 -23484.79} C_VEL
LIN {X 0,Y 154.676,Z 777.41,A -85,B 0,C 180,E1 -23488.407,E2 -23488.407} C_VEL
LIN {X 0,Y 154.905,Z 777.28,A -85,B 0,C 180,E1 -23492.603,E2 -23492.603} C_VEL
LIN {X 0,Y 155.664,Z 775.662,A -85,B 0,C 180,E1 -23497.787,E2 -23497.787} C_VEL
LIN {X 0,Y 156.85,Z 773.829,A -85,B 0,C 180,E1 -23501.307,E2 -23501.307} C_VEL
LIN {X 0,Y 158.312,Z 777.563,A -85,B 0,C 180,E1 -23505.45,E2 -23505.45} C_VEL
LIN {X 0,Y 159.695,Z 779.411,A -85,B 0,C 180,E1 -23507.945,E2 -23507.945} C_VEL
LIN {X 0,Y 161.47,Z 780.806,A -85,B 0,C 180,E1 -23510.379,E2 -23510.379} C_VEL
LIN {X 0,Y 166.132,Z 782.331,A -85,B 0,C 180,E1 -23515.028,E2 -23515.028} C_VEL
LIN {X 0,Y 169.139,Z 782.566,A -85,B 0,C 180,E1 -23517.2,E2 -23517.2} C_VEL
LIN {X 0,Y 176.087,Z 781.668,A -85,B 0,C 180,E1 -23521.258,E2 -23521.258} C_VEL
LIN {X 0,Y 180.04,Z 780.69,A -85,B 0,C 180,E1 -23523.129,E2 -23523.129} C_VEL
LIN {X 0,Y 184.209,Z 779.19,A -85,B 0,C 180,E1 -23524.912,E2 -23524.912} C_VEL
LIN {X 0,Y 193.333,Z 774.948,A -85,B 0,C 180,E1 -23528.171,E2 -23528.171} C_VEL
LIN {X 0,Y 200.767,Z 770.433,A -85,B 0,C 180,E1 -23530.363,E2 -23530.363} C_VEL
LIN {X 0,Y 208.704,Z 764.704,A -85,B 0,C 180,E1 -23532.339,E2 -23532.339} C_VEL
LIN {X 0,Y 217.564,Z 757.027,A -85,B 0,C 180,E1 -23534.201,E2 -23534.201} C_VEL
LIN {X 0,Y 224.662,Z 749.688,A -85,B 0,C 180,E1 -23535.516,E2 -23535.516} C_VEL
LIN {X 0,Y 225.8,Z 748.376,A -85,B 0,C 180,E1 -23535.716,E2 -23535.716} C_VEL
LIN {X 0,Y 217.553,Z 757.195,A -85,B 0,C 180,E1 -23537.281,E2 -23537.281} C_VEL
LIN {X 0,Y 209.175,Z 764.47,A -85,B 0,C 180,E1 -23539.067,E2 -23539.067} C_VEL
LIN {X 0,Y 201.232,Z 770.217,A -85,B 0,C 180,E1 -23541.049,E2 -23541.049} C_VEL
LIN {X 0,Y 196.182,Z 773.286,A -85,B 0,C 180,E1 -23542.482,E2 -23542.482} C_VEL
LIN {X 0,Y 189.851,Z 776.502,A -85,B 0,C 180,E1 -23544.531,E2 -23544.531} C_VEL
LIN {X 0,Y 186.787,Z 777.898,A -85,B 0,C 180,E1 -23545.64,E2 -23545.64} C_VEL
LIN {X 0,Y 182.441,Z 779.403,A -85,B 0,C 180,E1 -23547.363,E2 -23547.363} C_VEL
LIN {X 0,Y 174.563,Z 781.164,A -85,B 0,C 180,E1 -23551.11,E2 -23551.11} C_VEL
LIN {X 0,Y 171.098,Z 781.416,A -85,B 0,C 180,E1 -23553.138,E2 -23553.138} C_VEL
LIN {X 0,Y 165.12,Z 780.546,A -85,B 0,C 180,E1 -23557.476,E2 -23557.476} C_VEL
LIN {X 0,Y 162.729,Z 779.569,A -85,B 0,C 180,E1 -23559.787,E2 -23559.787} C_VEL
LIN {X 0,Y 160.704,Z 778.076,A -85,B 0,C 180,E1 -23562.174,E2 -23562.174} C_VEL
LIN {X 0,Y 157.874,Z 773.867,A -85,B 0,C 180,E1 -23567.139,E2 -23567.139} C_VEL
LIN {X 0,Y 156.9,Z 770.062,A -85,B 0,C 180,E1 -23570.534,E2 -23570.534} C_VEL
LIN {X 0,Y 156.595,Z 763.844,A -85,B 0,C 180,E1 -23574.85,E2 -23574.85} C_VEL
LIN {X 0,Y 156.774,Z 758.005,A -85,B 0,C 180,E1 -23578.073,E2 -23578.073} C_VEL
LIN {X 0,Y 157.166,Z 750.804,A -85,B 0,C 180,E1 -23581.281,E2 -23581.281} C_VEL
LIN {X 0,Y 157.466,Z 742.442,A -85,B 0,C 180,E1 -23584.159,E2 -23584.159} C_VEL
LIN {X 0,Y 157.824,Z 733.254,A -85,B 0,C 180,E1 -23586.713,E2 -23586.713} C_VEL
LIN {X 0,Y 158.259,Z 723.354,A -85,B 0,C 180,E1 -23588.942,E2 -23588.942} C_VEL
LIN {X 0,Y 158.718,Z 712.857,A -85,B 0,C 180,E1 -23590.763,E2 -23590.763} C_VEL
LIN {X 0,Y 159.094,Z 702.343,A -85,B 0,C 180,E1 -23592.139,E2 -23592.139} C_VEL
LIN {X 0,Y 159.797,Z 669.207,A -85,B 0,C 180,E1 -23595.164,E2 -23595.164} C_VEL
LIN {X 0,Y 160.086,Z 645.569,A -85,B 0,C 180,E1 -23597.197,E2 -23597.197} C_VEL
LIN {X 0,Y 158.569,Z 621.601,A -85,B 0,C 180,E1 -23599.163,E2 -23599.163} C_VEL
LIN {X 0,Y 158.471,Z 617.495,A -85,B 0,C 180,E1 -23599.596,E2 -23599.596} C_VEL
LIN {X 0,Y 160.858,Z 594.438,A -85,B 0,C 180,E1 -23607.307,E2 -23607.307} C_VEL
LIN {X 0,Y 161.852,Z 587.129,A -85,B 0,C 180,E1 -23609.718,E2 -23609.718} C_VEL
LIN {X 0,Y 160.542,Z 580.04,A -85,B 0,C 180,E1 -23612.302,E2 -23612.302} C_VEL
LIN {X 0,Y 160.555,Z 579.528,A -85,B 0,C 180,E1 -23613.08,E2 -23613.08} C_VEL
LIN {X 0,Y 161.851,Z 580.413,A -85,B 0,C 180,E1 -23614.012,E2 -23614.012} C_VEL
LIN {X 0,Y 163.857,Z 579.916,A -85,B 0,C 180,E1 -23615.009,E2 -23615.009} C_VEL
LIN {X 0,Y 165.449,Z 579.212,A -85,B 0,C 180,E1 -23615.744,E2 -23615.744} C_VEL
LIN {X 0,Y 168.126,Z 579.588,A -85,B 0,C 180,E1 -23617.029,E2 -23617.029} C_VEL
LIN {X 0,Y 172.72,Z 586.157,A -85,B 0,C 180,E1 -23619.445,E2 -23619.445} C_VEL
LIN {X 0,Y 177.601,Z 593.418,A -85,B 0,C 180,E1 -23621.772,E2 -23621.772} C_VEL
LIN {X 0,Y 183.367,Z 602.858,A -85,B 0,C 180,E1 -23624.29,E2 -23624.29} C_VEL
LIN {X 0,Y 186.816,Z 609.356,A -85,B 0,C 180,E1 -23625.716,E2 -23625.716} C_VEL
LIN {X 0,Y 191.314,Z 620.162,A -85,B 0,C 180,E1 -23627.569,E2 -23627.569} C_VEL
LIN {X 0,Y 188.534,Z 665.522,A -85,B 0,C 180,E1 -23629.157,E2 -23629.157} C_VEL
LIN {X 0,Y 186.844,Z 678.933,A -85,B 0,C 180,E1 -23629.993,E2 -23629.993} C_VEL
LIN {X 0,Y 184.442,Z 691.881,A -85,B 0,C 180,E1 -23631.218,E2 -23631.218} C_VEL
LIN {X 0,Y 181.511,Z 703.66,A -85,B 0,C 180,E1 -23632.77,E2 -23632.77} C_VEL
LIN {X 0,Y 178.096,Z 714.99,A -85,B 0,C 180,E1 -23634.749,E2 -23634.749} C_VEL
LIN {X 0,Y 174.472,Z 725.2,A -85,B 0,C 180,E1 -23637.055,E2 -23637.055} C_VEL
LIN {X 0,Y 170.777,Z 734.52,A -85,B 0,C 180,E1 -23639.794,E2 -23639.794} C_VEL
LIN {X 0,Y 167.022,Z 743.254,A -85,B 0,C 180,E1 -23643.104,E2 -23643.104} C_VEL
LIN {X 0,Y 163.541,Z 750.418,A -85,B 0,C 180,E1 -23646.575,E2 -23646.575} C_VEL
LIN {X 0,Y 161.081,Z 755.248,A -85,B 0,C 180,E1 -23649.569,E2 -23649.569} C_VEL
LIN {X 0,Y 158.73,Z 759.937,A -85,B 0,C 180,E1 -23653.272,E2 -23653.272} C_VEL
LIN {X 0,Y 156.934,Z 763.518,A -85,B 0,C 180,E1 -23657.059,E2 -23657.059} C_VEL
LIN {X 0,Y 156.087,Z 765.366,A -85,B 0,C 180,E1 -23659.622,E2 -23659.622} C_VEL
LIN {X 0,Y 155.507,Z 766.754,A -85,B 0,C 180,E1 -23662.206,E2 -23662.206} C_VEL
LIN {X 0,Y 154.905,Z 768.348,A -85,B 0,C 180,E1 -23667.397,E2 -23667.397} C_VEL
LIN {X 0,Y 154.861,Z 768.575,A -85,B 0,C 180,E1 -23669.998,E2 -23669.998} C_VEL
LIN {X 0,Y 154.952,Z 768.169,A -85,B 0,C 180,E1 -23673.769,E2 -23673.769} C_VEL
LIN {X 0,Y 155.505,Z 766.831,A -85,B 0,C 180,E1 -23677.79,E2 -23677.79} C_VEL
LIN {X 0,Y 156.085,Z 765.476,A -85,B 0,C 180,E1 -23680.374,E2 -23680.374} C_VEL
LIN {X 0,Y 157.443,Z 762.606,A -85,B 0,C 180,E1 -23684.21,E2 -23684.21} C_VEL
LIN {X 0,Y 159.421,Z 758.71,A -85,B 0,C 180,E1 -23687.972,E2 -23687.972} C_VEL
LIN {X 0,Y 161.952,Z 753.689,A -85,B 0,C 180,E1 -23691.643,E2 -23691.643} C_VEL
LIN {X 0,Y 165.13,Z 747.358,A -85,B 0,C 180,E1 -23695.186,E2 -23695.186} C_VEL
LIN {X 0,Y 168.756,Z 739.634,A -85,B 0,C 180,E1 -23698.522,E2 -23698.522} C_VEL
LIN {X 0,Y 172.098,Z 731.543,A -85,B 0,C 180,E1 -23701.306,E2 -23701.306} C_VEL
LIN {X 0,Y 175.936,Z 721.508,A -85,B 0,C 180,E1 -23704.001,E2 -23704.001} C_VEL
LIN {X 0,Y 179.724,Z 710.403,A -85,B 0,C 180,E1 -23706.257,E2 -23706.257} C_VEL
LIN {X 0,Y 182.822,Z 699.511,A -85,B 0,C 180,E1 -23707.954,E2 -23707.954} C_VEL
LIN {X 0,Y 185.536,Z 687.461,A -85,B 0,C 180,E1 -23709.379,E2 -23709.379} C_VEL
LIN {X 0,Y 187.607,Z 674.86,A -85,B 0,C 180,E1 -23710.447,E2 -23710.447} C_VEL
LIN {X 0,Y 189.067,Z 661.416,A -85,B 0,C 180,E1 -23711.145,E2 -23711.145} C_VEL
LIN {X 0,Y 191.474,Z 620.403,A -85,B 0,C 180,E1 -23712.556,E2 -23712.556} C_VEL
LIN {X 0,Y 186.101,Z 607.602,A -85,B 0,C 180,E1 -23714.784,E2 -23714.784} C_VEL
LIN {X 0,Y 180.158,Z 597.417,A -85,B 0,C 180,E1 -23717.289,E2 -23717.289} C_VEL
LIN {X 0,Y 173.979,Z 587.868,A -85,B 0,C 180,E1 -23720.159,E2 -23720.159} C_VEL
LIN {X 0,Y 170.639,Z 583.177,A -85,B 0,C 180,E1 -23721.844,E2 -23721.844} C_VEL
LIN {X 0,Y 168.182,Z 579.695,A -85,B 0,C 180,E1 -23723.173,E2 -23723.173} C_VEL
LIN {X 0,Y 165.464,Z 575.897,A -85,B 0,C 180,E1 -23724.738,E2 -23724.738} C_VEL
LIN {X 0,Y 162.368,Z 572.445,A -85,B 0,C 180,E1 -23726.597,E2 -23726.597} C_VEL
LIN {X 0,Y 161.266,Z 570.418,A -85,B 0,C 180,E1 -23727.363,E2 -23727.363} C_VEL
LIN {X 0,Y 158.941,Z 568.521,A -85,B 0,C 180,E1 -23728.869,E2 -23728.869} C_VEL
LIN {X 0,Y 157.608,Z 566.244,A -85,B 0,C 180,E1 -23729.89,E2 -23729.89} C_VEL
LIN {X 0,Y 157.283,Z 564.891,A -85,B 0,C 180,E1 -23730.283,E2 -23730.283} C_VEL
LIN {X 0,Y 157.316,Z 564.877,A -85,B 0,C 180,E1 -23733.465,E2 -23733.465} C_VEL
LIN {X 0,Y 157.39,Z 564.87,A -85,B 0,C 180,E1 -23739.665,E2 -23739.665} C_VEL
LIN {X 0,Y 157.463,Z 564.85,A -85,B 0,C 180,E1 -23744.467,E2 -23744.467} C_VEL
LIN {X 0,Y 157.723,Z 564.815,A -85,B 0,C 180,E1 -23749.733,E2 -23749.733} C_VEL
LIN {X 0,Y 157.805,Z 564.818,A -85,B 0,C 180,E1 -23752.322,E2 -23752.322} C_VEL
LIN {X 0,Y 158.253,Z 564.773,A -85,B 0,C 180,E1 -23760,E2 -23760} C_VEL
LIN {X 0,Y 157.818,Z 564.822,A -85,B 0,C 180,E1 -23767.677,E2 -23767.677} C_VEL
LIN {X 0,Y 157.699,Z 564.824,A -85,B 0,C 180,E1 -23771.361,E2 -23771.361} C_VEL
LIN {X 0,Y 157.463,Z 564.852,A -85,B 0,C 180,E1 -23775.533,E2 -23775.533} C_VEL
LIN {X 0,Y 157.365,Z 564.869,A -85,B 0,C 180,E1 -23780.933,E2 -23780.933} C_VEL
LIN {X 0,Y 157.308,Z 564.877,A -85,B 0,C 180,E1 -23786.685,E2 -23786.685} C_VEL
LIN {X 0,Y 157.285,Z 564.891,A -85,B 0,C 180,E1 -23789.348,E2 -23789.348} C_VEL
LIN {X 0,Y 158.226,Z 567.611,A -85,B 0,C 180,E1 -23790.256,E2 -23790.256} C_VEL
LIN {X 0,Y 160.375,Z 569.876,A -85,B 0,C 180,E1 -23791.727,E2 -23791.727} C_VEL
LIN {X 0,Y 161.465,Z 570.663,A -85,B 0,C 180,E1 -23792.406,E2 -23792.406} C_VEL
LIN {X 0,Y 163.42,Z 573.892,A -85,B 0,C 180,E1 -23793.714,E2 -23793.714} C_VEL
LIN {X 0,Y 165.554,Z 576.058,A -85,B 0,C 180,E1 -23794.958,E2 -23794.958} C_VEL
LIN {X 0,Y 169.847,Z 582.804,A -85,B 0,C 180,E1 -23797.427,E2 -23797.427} C_VEL
LIN {X 0,Y 173.539,Z 588.858,A -85,B 0,C 180,E1 -23799.369,E2 -23799.369} C_VEL
LIN {X 0,Y 178.236,Z 597.304,A -85,B 0,C 180,E1 -23801.666,E2 -23801.666} C_VEL
LIN {X 0,Y 183.494,Z 608.039,A -85,B 0,C 180,E1 -23804.061,E2 -23804.061} C_VEL
LIN {X 0,Y 188.926,Z 621.181,A -85,B 0,C 180,E1 -23806.405,E2 -23806.405} C_VEL
LIN {X 0,Y 190.741,Z 626.334,A -85,B 0,C 180,E1 -23807.177,E2 -23807.177} C_VEL
LIN {X 0,Y 190.944,Z 630.401,A -85,B 0,C 180,E1 -23807.437,E2 -23807.437} C_VEL
LIN {X 0,Y 188.195,Z 673.96,A -85,B 0,C 180,E1 -23808.951,E2 -23808.951} C_VEL
LIN {X 0,Y 186.387,Z 687.604,A -85,B 0,C 180,E1 -23809.793,E2 -23809.793} C_VEL
LIN {X 0,Y 183.867,Z 699.914,A -85,B 0,C 180,E1 -23810.902,E2 -23810.902} C_VEL
LIN {X 0,Y 180.575,Z 712.584,A -85,B 0,C 180,E1 -23812.549,E2 -23812.549} C_VEL
LIN {X 0,Y 177.203,Z 723.31,A -85,B 0,C 180,E1 -23814.405,E2 -23814.405} C_VEL
LIN {X 0,Y 175.073,Z 728.104,A -85,B 0,C 180,E1 -23815.289,E2 -23815.289} C_VEL
LIN {X 0,Y 169.8,Z 735.552,A -85,B 0,C 180,E1 -23816.586,E2 -23816.586} C_VEL
LIN {X 0,Y 164.288,Z 742.45,A -85,B 0,C 180,E1 -23818.145,E2 -23818.145} C_VEL
LIN {X 0,Y 161.84,Z 746.382,A -85,B 0,C 180,E1 -23819.436,E2 -23819.436} C_VEL
LIN {X 0,Y 157.769,Z 755.014,A -85,B 0,C 180,E1 -23823.182,E2 -23823.182} C_VEL
LIN {X 0,Y 154.178,Z 762.067,A -85,B 0,C 180,E1 -23827.206,E2 -23827.206} C_VEL
LIN {X 0,Y 151.55,Z 767.168,A -85,B 0,C 180,E1 -23831.06,E2 -23831.06} C_VEL
LIN {X 0,Y 149.63,Z 771.139,A -85,B 0,C 180,E1 -23835.031,E2 -23835.031} C_VEL
LIN {X 0,Y 148.391,Z 774.078,A -85,B 0,C 180,E1 -23839.082,E2 -23839.082} C_VEL
LIN {X 0,Y 147.898,Z 775.475,A -85,B 0,C 180,E1 -23841.807,E2 -23841.807} C_VEL
LIN {X 0,Y 147.634,Z 776.474,A -85,B 0,C 180,E1 -23844.539,E2 -23844.539} C_VEL
LIN {X 0,Y 147.606,Z 777.254,A -85,B 0,C 180,E1 -23849.112,E2 -23849.112} C_VEL
LIN {X 0,Y 147.91,Z 776.888,A -85,B 0,C 180,E1 -23853.781,E2 -23853.781} C_VEL
LIN {X 0,Y 148.641,Z 775.458,A -85,B 0,C 180,E1 -23858.157,E2 -23858.157} C_VEL
LIN {X 0,Y 150.372,Z 772.997,A -85,B 0,C 180,E1 -23862.829,E2 -23862.829} C_VEL
LIN {X 0,Y 151.612,Z 776.15,A -85,B 0,C 180,E1 -23866.151,E2 -23866.151} C_VEL
LIN {X 0,Y 154.905,Z 779.744,A -85,B 0,C 180,E1 -23871.284,E2 -23871.284} C_VEL
LIN {X 0,Y 157.064,Z 781.045,A -85,B 0,C 180,E1 -23873.75,E2 -23873.75} C_VEL
LIN {X 0,Y 159.745,Z 781.856,A -85,B 0,C 180,E1 -23876.103,E2 -23876.103} C_VEL
LIN {X 0,Y 166.315,Z 782.442,A -85,B 0,C 180,E1 -23880.472,E2 -23880.472} C_VEL
LIN {X 0,Y 170.075,Z 782.105,A -85,B 0,C 180,E1 -23882.495,E2 -23882.495} C_VEL
LIN {X 0,Y 178.499,Z 780.254,A -85,B 0,C 180,E1 -23886.201,E2 -23886.201} C_VEL
LIN {X 0,Y 185.469,Z 777.779,A -85,B 0,C 180,E1 -23888.702,E2 -23888.702} C_VEL
LIN {X 0,Y 192.953,Z 774.27,A -85,B 0,C 180,E1 -23890.969,E2 -23890.969} C_VEL
LIN {X 0,Y 200.985,Z 769.644,A -85,B 0,C 180,E1 -23892.992,E2 -23892.992} C_VEL
LIN {X 0,Y 209.449,Z 763.759,A -85,B 0,C 180,E1 -23894.803,E2 -23894.803} C_VEL
LIN {X 0,Y 213.409,Z 760.574,A -85,B 0,C 180,E1 -23895.567,E2 -23895.567} C_VEL
LIN {X 0,Y 212.674,Z 761.208,A -85,B 0,C 180,E1 -23896.055,E2 -23896.055} C_VEL
LIN {X 0,Y 204.091,Z 767.724,A -85,B 0,C 180,E1 -23897.817,E2 -23897.817} C_VEL
LIN {X 0,Y 195.922,Z 772.688,A -85,B 0,C 180,E1 -23899.783,E2 -23899.783} C_VEL
LIN {X 0,Y 188.234,Z 776.442,A -85,B 0,C 180,E1 -23901.971,E2 -23901.971} C_VEL
LIN {X 0,Y 181.03,Z 779.103,A -85,B 0,C 180,E1 -23904.385,E2 -23904.385} C_VEL
LIN {X 0,Y 176.541,Z 780.326,A -85,B 0,C 180,E1 -23906.129,E2 -23906.129} C_VEL
LIN {X 0,Y 172.313,Z 781.154,A -85,B 0,C 180,E1 -23907.98,E2 -23907.98} C_VEL
LIN {X 0,Y 168.384,Z 781.439,A -85,B 0,C 180,E1 -23909.943,E2 -23909.943} C_VEL
LIN {X 0,Y 161.6,Z 780.924,A -85,B 0,C 180,E1 -23914.221,E2 -23914.221} C_VEL
LIN {X 0,Y 158.619,Z 779.997,A -85,B 0,C 180,E1 -23916.499,E2 -23916.499} C_VEL
LIN {X 0,Y 154.045,Z 776.966,A -85,B 0,C 180,E1 -23921.376,E2 -23921.376} C_VEL
LIN {X 0,Y 151.754,Z 773.604,A -85,B 0,C 180,E1 -23925.243,E2 -23925.243} C_VEL
LIN {X 0,Y 150.44,Z 769.175,A -85,B 0,C 180,E1 -23929.23,E2 -23929.23} C_VEL
LIN {X 0,Y 149.903,Z 763.598,A -85,B 0,C 180,E1 -23933.269,E2 -23933.269} C_VEL
LIN {X 0,Y 150.03,Z 757.809,A -85,B 0,C 180,E1 -23936.643,E2 -23936.643} C_VEL
LIN {X 0,Y 150.4,Z 750.692,A -85,B 0,C 180,E1 -23940,E2 -23940} C_VEL
LIN {X 0,Y 150.733,Z 742.596,A -85,B 0,C 180,E1 -23943.007,E2 -23943.007} C_VEL
LIN {X 0,Y 150.926,Z 734.769,A -85,B 0,C 180,E1 -23945.344,E2 -23945.344} C_VEL
LIN {X 0,Y 151.357,Z 725.234,A -85,B 0,C 180,E1 -23947.672,E2 -23947.672} C_VEL
LIN {X 0,Y 151.896,Z 712.925,A -85,B 0,C 180,E1 -23949.992,E2 -23949.992} C_VEL
LIN {X 0,Y 152.199,Z 702.077,A -85,B 0,C 180,E1 -23951.487,E2 -23951.487} C_VEL
LIN {X 0,Y 152.718,Z 672.407,A -85,B 0,C 180,E1 -23954.399,E2 -23954.399} C_VEL
LIN {X 0,Y 153.07,Z 645.725,A -85,B 0,C 180,E1 -23956.848,E2 -23956.848} C_VEL
LIN {X 0,Y 151.504,Z 621.679,A -85,B 0,C 180,E1 -23958.905,E2 -23958.905} C_VEL
LIN {X 0,Y 151.419,Z 617.664,A -85,B 0,C 180,E1 -23959.312,E2 -23959.312} C_VEL
LIN {X 0,Y 153.939,Z 592.985,A -85,B 0,C 180,E1 -23967.902,E2 -23967.902} C_VEL
LIN {X 0,Y 154.683,Z 588.468,A -85,B 0,C 180,E1 -23969.705,E2 -23969.705} C_VEL
LIN {X 0,Y 154.941,Z 587.734,A -85,B 0,C 180,E1 -23970.403,E2 -23970.403} C_VEL
LIN {X 0,Y 155.638,Z 588.418,A -85,B 0,C 180,E1 -23971.134,E2 -23971.134} C_VEL
LIN {X 0,Y 157.134,Z 588.525,A -85,B 0,C 180,E1 -23972.044,E2 -23972.044} C_VEL
LIN {X 0,Y 159.368,Z 587.008,A -85,B 0,C 180,E1 -23973.193,E2 -23973.193} C_VEL
LIN {X 0,Y 161.595,Z 587.506,A -85,B 0,C 180,E1 -23974.43,E2 -23974.43} C_VEL
LIN {X 0,Y 164.494,Z 586.594,A -85,B 0,C 180,E1 -23975.821,E2 -23975.821} C_VEL
LIN {X 0,Y 165.998,Z 586.587,A -85,B 0,C 180,E1 -23976.54,E2 -23976.54} C_VEL
LIN {X 0,Y 171.534,Z 594.788,A -85,B 0,C 180,E1 -23979.52,E2 -23979.52} C_VEL
LIN {X 0,Y 178.011,Z 605.275,A -85,B 0,C 180,E1 -23982.621,E2 -23982.621} C_VEL
LIN {X 0,Y 182.43,Z 613.541,A -85,B 0,C 180,E1 -23984.577,E2 -23984.577} C_VEL
LIN {X 0,Y 186.01,Z 622.284,A -85,B 0,C 180,E1 -23986.156,E2 -23986.156} C_VEL
LIN {X 0,Y 183.225,Z 665.741,A -85,B 0,C 180,E1 -23987.705,E2 -23987.705} C_VEL
LIN {X 0,Y 181.528,Z 678.872,A -85,B 0,C 180,E1 -23988.537,E2 -23988.537} C_VEL
LIN {X 0,Y 179.216,Z 691.013,A -85,B 0,C 180,E1 -23989.678,E2 -23989.678} C_VEL
LIN {X 0,Y 176.439,Z 702.287,A -85,B 0,C 180,E1 -23991.142,E2 -23991.142} C_VEL
LIN {X 0,Y 172.779,Z 713.911,A -85,B 0,C 180,E1 -23993.13,E2 -23993.13} C_VEL
LIN {X 0,Y 168.959,Z 724.353,A -85,B 0,C 180,E1 -23995.474,E2 -23995.474} C_VEL
LIN {X 0,Y 164.95,Z 734.119,A -85,B 0,C 180,E1 -23998.339,E2 -23998.339} C_VEL
LIN {X 0,Y 161.348,Z 742.115,A -85,B 0,C 180,E1 -24001.369,E2 -24001.369} C_VEL
LIN {X 0,Y 157.659,Z 749.514,A -85,B 0,C 180,E1 -24004.943,E2 -24004.943} C_VEL
LIN {X 0,Y 154.433,Z 755.455,A -85,B 0,C 180,E1 -24008.648,E2 -24008.648} C_VEL
LIN {X 0,Y 151.953,Z 760.142,A -85,B 0,C 180,E1 -24012.502,E2 -24012.502} C_VEL
LIN {X 0,Y 150.019,Z 763.724,A -85,B 0,C 180,E1 -24016.451,E2 -24016.451} C_VEL
LIN {X 0,Y 149.113,Z 765.572,A -85,B 0,C 180,E1 -24019.131,E2 -24019.131} C_VEL
LIN {X 0,Y 148.47,Z 766.959,A -85,B 0,C 180,E1 -24021.834,E2 -24021.834} C_VEL
LIN {X 0,Y 147.855,Z 768.43,A -85,B 0,C 180,E1 -24026.565,E2 -24026.565} C_VEL
LIN {X 0,Y 147.766,Z 768.78,A -85,B 0,C 180,E1 -24029.998,E2 -24029.998} C_VEL
LIN {X 0,Y 147.839,Z 768.479,A -85,B 0,C 180,E1 -24033.335,E2 -24033.335} C_VEL
LIN {X 0,Y 148.468,Z 767.035,A -85,B 0,C 180,E1 -24038.162,E2 -24038.162} C_VEL
LIN {X 0,Y 149.11,Z 765.68,A -85,B 0,C 180,E1 -24040.865,E2 -24040.865} C_VEL
LIN {X 0,Y 150.572,Z 762.809,A -85,B 0,C 180,E1 -24044.873,E2 -24044.873} C_VEL
LIN {X 0,Y 152.693,Z 758.913,A -85,B 0,C 180,E1 -24048.793,E2 -24048.793} C_VEL
LIN {X 0,Y 155.379,Z 753.892,A -85,B 0,C 180,E1 -24052.608,E2 -24052.608} C_VEL
LIN {X 0,Y 158.746,Z 747.561,A -85,B 0,C 180,E1 -24056.275,E2 -24056.275} C_VEL
LIN {X 0,Y 162.416,Z 740.112,A -85,B 0,C 180,E1 -24059.612,E2 -24059.612} C_VEL
LIN {X 0,Y 166.156,Z 731.568,A -85,B 0,C 180,E1 -24062.632,E2 -24062.632} C_VEL
LIN {X 0,Y 170.103,Z 721.709,A -85,B 0,C 180,E1 -24065.337,E2 -24065.337} C_VEL
LIN {X 0,Y 174.054,Z 710.603,A -85,B 0,C 180,E1 -24067.639,E2 -24067.639} C_VEL
LIN {X 0,Y 177.291,Z 699.71,A -85,B 0,C 180,E1 -24069.362,E2 -24069.362} C_VEL
LIN {X 0,Y 180.123,Z 687.658,A -85,B 0,C 180,E1 -24070.807,E2 -24070.807} C_VEL
LIN {X 0,Y 182.271,Z 675.046,A -85,B 0,C 180,E1 -24071.894,E2 -24071.894} C_VEL
LIN {X 0,Y 183.804,Z 661.271,A -85,B 0,C 180,E1 -24072.615,E2 -24072.615} C_VEL
LIN {X 0,Y 186.188,Z 622.574,A -85,B 0,C 180,E1 -24073.964,E2 -24073.964} C_VEL
LIN {X 0,Y 181.675,Z 611.753,A -85,B 0,C 180,E1 -24075.963,E2 -24075.963} C_VEL
LIN {X 0,Y 175.401,Z 600.795,A -85,B 0,C 180,E1 -24078.805,E2 -24078.805} C_VEL
LIN {X 0,Y 170.127,Z 592.607,A -85,B 0,C 180,E1 -24081.433,E2 -24081.433} C_VEL
LIN {X 0,Y 165.142,Z 585.432,A -85,B 0,C 180,E1 -24084.194,E2 -24084.194} C_VEL
LIN {X 0,Y 162.074,Z 581.252,A -85,B 0,C 180,E1 -24086.061,E2 -24086.061} C_VEL
LIN {X 0,Y 159.438,Z 578,A -85,B 0,C 180,E1 -24087.775,E2 -24087.775} C_VEL
LIN {X 0,Y 158.547,Z 576.618,A -85,B 0,C 180,E1 -24088.411,E2 -24088.411} C_VEL
LIN {X 0,Y 155.998,Z 573.951,A -85,B 0,C 180,E1 -24090.222,E2 -24090.222} C_VEL
LIN {X 0,Y 154.688,Z 571.494,A -85,B 0,C 180,E1 -24091.321,E2 -24091.321} C_VEL
LIN {X 0,Y 152.117,Z 569.719,A -85,B 0,C 180,E1 -24093.343,E2 -24093.343} C_VEL
LIN {X 0,Y 150.618,Z 567.322,A -85,B 0,C 180,E1 -24094.775,E2 -24094.775} C_VEL
